METHOD OutputPublish
  VAR_INPUT
    PayloadSize : UDINT;
    PayloadPos : POINTER TO BYTE;  (* be aware, don't use network buffer, IP_CONTROL may change content *)
    TopicSize : UDINT;
    TopicPos : POINTER TO BYTE;  (* be aware, don't use network buffer, IP_CONTROL may change content, must be zero terminated! *)
    MQTT_IN_OUT : POINTER TO MQTT_IN_OUT;
  END_VAR
  VAR
    i : UINT;
    match : TOPIC_MATCH;
    PointerToSplit : POINTER TO SPLIT_TOPIC;
    DataForCallback : CALLBACK_DATA;
  END_VAR
                  //here make everything to give out publish, and test if topic fits to my borders...
CountOutputPublishCalled := CountOutputPublishCalled + 1;
IF MySplitTopic.NewTopic(in:= TopicPos, test := FALSE, SizeOfString:= UDINT_TO_UINT(TopicSize)) = TOPIC_VALID.TOPIC_NOT_VALID THEN
	//topic is not in my borders so throw away data...
	{info 'configure to disconnect?'}
	{ info 'make count var...'}
	CountSplitTopicSizeExceeded := CountSplitTopicSizeExceeded + 1;
	RETURN;
END_IF
//now search the right callback and call it...
PointerToSplit := MySplitTopic.GetSplitTopic();
DataForCallback.Payload := PayloadPos;
DataForCallback.PayloadSize := PayloadSize;
DataForCallback.PayloadString :=PayloadPos;
DataForCallback.TopicOut := TopicPos;
DataForCallback.TopicOutSplit := PointerToSplit;
DataForCallback.PayloadIsString := SubscribeCallbacks[i].ExpectingString;

FOR i := 0 TO CALLBACKS_BUFFER_SIZE - 1 DO
	IF NOT SubscribeCallbacks[i].free THEN
		match := SubscribeCallbacks[i].SplitTopic^.CheckTopicMatchToMe(with:=PointerToSplit);
		IF match = TOPIC_MATCH.TOPIC_MATCHES THEN
			SubscribeCallbacks[i].Callback.PublishRecived(Data:=DataForCallback);
		END_IF
	END_IF
END_FOR


                
END_METHOD

METHOD MergeSplitedPublish
  VAR_INPUT
    MQTT_IN_OUT : POINTER TO MQTT_IN_OUT;
  END_VAR
  VAR
    BytesToMove : UINT;
  END_VAR
                  //move every new data to publish recive buffer untill all data is recived
BytesToMove := TO_UINT(MIN(com.R_BUF.SIZE, SplitPublishLength - SplitPublishBufferSize));
MEM.MemMove(pSource:= ADR(COM.R_BUF.BUFFER), pDestination:= ADR(SplitPublishBuffer[SplitPublishBufferSize]), uiNumberOfBytes:= BytesToMove);
SplitPublishBufferSize := SplitPublishBufferSize + BytesToMove;
IF SplitPublishBufferSize >= SplitPublishLength THEN
	//SplitPublishLock := TRUE;
	PublishSplited := FALSE;
	//ParsePublish will insert string termination if no network buffer
	ParseIncomingPublish(
	MQTT_IN_OUT:= MQTT_IN_OUT, 
	idx:= 0, 
	BufferIn:= SplitPublishBuffer, 
	BufferSize:= SplitPublishBufferSize,
	NetworkBuffer := FALSE);
END_IF
//check if there is more data in buffer --> new packet
IF BytesToMove < COM.R_BUF.SIZE THEN
	//move buffer and set new size...
	MEM.MemMove(pSource:= ADR(COM.R_BUF.BUFFER[BytesToMove]), pDestination:= ADR(COM.R_BUF.BUFFER),
				uiNumberOfBytes:= COM.R_BUF.SIZE - BytesToMove);
	COM.R_BUF.SIZE := COM.R_BUF.SIZE - BytesToMove;
ELSE
	//clear buffer
	COM.R_BUF.SIZE := 0;
	COM.MQTT_RCV_STATE := BYTE#0;//recive zurücksetzten	
END_IF
                
END_METHOD

METHOD Publish : BOOL
  VAR_INPUT
    data : POINTER TO DATA_TO_BROKER;
  END_VAR
  VAR
    i : UINT;
  END_VAR
                  Publish := FALSE;
FOR i := 0 TO MyConstants.QoS_BUFFER_SIZE - 1 DO
	IF OutData[i].step = STEPS_OUT.WAIT_DATA THEN
		OutData[i].InDataFromFb := data;//set Data
		//Pakte id = slot + 1....
		OutData[i].InDataFromFb^.PaketId := i + 1;
		OutgoingPublishOrderIndexCounter := OutgoingPublishOrderIndexCounter + 1;
		OutData[i].PUBLISHOrder :=  OutgoingPublishOrderIndexCounter;
		OutData[i].step := STEPS_OUT.SEND_PUBLSIH;
		CountSendedPublishs := CountSendedPublishs + 1;
		CounterPublishSendForMonitor := CounterPublishSendForMonitor + 1;
		OutData[i].PUBRELRepeatCounter := 0;
		Publish := TRUE;
		EXIT;
	END_IF
END_FOR
                
END_METHOD

METHOD PublishSendDone
  VAR_INPUT
    slot : POINTER TO MQTT_OUT_DATA;
  END_VAR
                  slot^.TimeOutStarted := TRUE;//start Timeout
CASE slot^.InDataFromFb^.MessageQoS OF
	QoS.AtMostOnce:
	//paket gone and bye bye, on QoS 0 
	slot^.InDataFromFb^.SendSucsess := TRUE;
	slot^.step := STEPS_OUT.WAIT_DATA;//can get new data
	QoS.AtLeastOnce:
		slot^.step := STEPS_OUT.WAIT_PUBACK;//wait for ACK
		IF NOT slot^.InDataFromFb^.DUP THEN
			Publishsunacknowledged := Publishsunacknowledged + 1;
		END_IF
	QoS.ExactlyOnce:
		slot^.step := STEPS_OUT.WAIT_PUBREC;//wait for REC
		IF NOT slot^.InDataFromFb^.DUP THEN
			Publishsunacknowledged := Publishsunacknowledged + 1;
		END_IF
END_CASE
                
END_METHOD
END_FUNCTION_BLOCK

FUNCTION_BLOCK HandleSplitTopic
  VAR
    MySplitTopic : SPLIT_TOPIC;
    InitFull : BOOL;
    InitLow : BOOL;
    SplitLength : POINTER TO UINT;  (* this is going to be a pointer to a array of uint to store the string length(and so memmory size) in the string array *)
    TopicsLevel : UINT;
    SplitElementSize : UINT;
    CountSizeExceeded : ULINT;
    TopicsIndexMax : UINT;
    dynMemUsage : POINTER TO UDINT;
  END_VAR

            {info 'TODO test of zeros in strings'}
          

(* use FOR high change OF topic, needs more ram, saves TIME... allocates all memory for the string arrays and strings usefull for often changed topics like recive publish *)
METHOD FullInit : BOOL
  VAR_INPUT
    TopicsLevelInit : UINT;
    SplitElementSizeInit : UINT;
    dynMemUsageInit : POINTER TO UDINT;
  END_VAR
  VAR
    iu : UINT;
  END_VAR
                  dynMemUsage := dynMemUsageInit;
destroy();

InitFull := TRUE;
InitLow := FALSE;

TopicsLevel := TopicsLevelInit;
SplitElementSize := SplitElementSizeInit + 1;//add 1 for trailing 0
IF TopicsLevel > 0 THEN
	TopicsIndexMax := TopicsLevel - 1;
ELSE
	TopicsIndexMax := 0;
END_IF

{warning disable C0033}
//get memory for array of pointer to strings
//MySplitTopic.Topics := SysMem23.SysMemAlloc(dwSize:= TopicsLevel * SIZEOF(MySplitTopic.Topics^));
{info 'semaphore'}
MySplitTopic.Topics := __NEW(POINTER TO STRING, TopicsLevel);
dynMemUsage^ := dynMemUsage^ + TopicsLevel * SIZEOF(MySplitTopic.Topics^);
FOR iu := 0 TO TopicsLevel - 1 DO
	//Get memory for strings
	//MySplitTopic.Topics[iu] := SysMem23.SysMemAlloc(dwSize:= SplitElementSize);	
	{info 'semaphore'}
	MySplitTopic.Topics[iu] := __NEW(BYTE, SplitElementSize);	
	dynMemUsage^ := dynMemUsage^ + SplitElementSize;
END_FOR
{warning restore C0033}

                
END_METHOD

(* use for low change of topic, saves mem, needs time dynamic allocation of memory, usefull for static stopis like compare of subscription topic *)
METHOD LowInit : BOOL
  VAR_INPUT
    TopicsLevelInit : UINT;
    SplitElementSizeInit : UINT;
    dynMemUsageInit : POINTER TO UDINT;
  END_VAR
  VAR
    iu : UINT;
  END_VAR
                  dynMemUsage := dynMemUsageInit;
destroy();
InitFull := FALSE;
InitLow := TRUE;

TopicsLevel := TopicsLevelInit;
SplitElementSize :=SplitElementSizeInit;
IF TopicsLevel > 0 THEN
	TopicsIndexMax := TopicsLevel - 1;
ELSE
	TopicsIndexMax := 0;
END_IF
{warning disable C0033}
//get memory for array of pointer to string 

//MySplitTopic.Topics := SysMem23.SysMemAlloc(dwSize:= TopicsLevel * SIZEOF(MySplitTopic.Topics^));
MySplitTopic.Topics := __NEW(POINTER TO STRING, TopicsLevel);
{info 'semaphore'}
dynMemUsage^ := dynMemUsage^ + TopicsLevel * SIZEOF(MySplitTopic.Topics^);
//get memory for array of length of strings
//SplitLength := SysMem23.SysMemAlloc(dwSize:= TopicsLevel * SIZEOF(SplitLength^));
{info 'semaphore'}
SplitLength := __NEW(POINTER TO STRING, TopicsLevel);
dynMemUsage^ := dynMemUsage^ + TopicsLevel * SIZEOF(SplitLength^);
{warning restore C0033}

                
END_METHOD

METHOD destroy : BOOL
  VAR
    iu : UINT;
  END_VAR
                  GVL_MQTT.ProgNum := PROG_NUM.DESTROY_SPLIT_TOPIC;
IF InitFull THEN
{warning disable C0033}
	FOR iu := 0 TO TopicsLevel - 1 DO
		{info 'semaphore'}
		//SysMem23.SysMemFree(dwAddress:= MySplitTopic.Topics[iu], dwSize:= SplitElementSize);
		__DELETE(MySplitTopic.Topics[iu]);
		dynMemUsage^ := dynMemUsage^ - SplitElementSize;
	END_FOR
	{info 'semaphore'}
	//SysMem23.SysMemFree(dwAddress:= MySplitTopic.Topics, dwSize:= TopicsLevel * SIZEOF(MySplitTopic.Topics^));
	__DELETE(MySplitTopic.Topics);
	dynMemUsage^ := dynMemUsage^ - (TopicsLevel * SIZEOF(MySplitTopic.Topics^));
	InitFull := FALSE;
END_IF

IF InitLow THEN
	DestroyOldSplit();
	{info 'semaphore'}
	//SysMem23.SysMemFree(dwAddress:= MySplitTopic.Topics, dwSize:= TopicsLevel * SIZEOF(MySplitTopic.Topics^));
	__DELETE(MySplitTopic.Topics);
	dynMemUsage^ := dynMemUsage^ - (TopicsLevel * SIZEOF(MySplitTopic.Topics^));
	//SysMem23.SysMemFree(dwAddress:= SplitLength, dwSize:= TopicsLevel * SIZEOF(SplitLength^));
	{info 'semaphore'}
	//SysMem.SysMemFreeData(pMemory:= SplitLength, dwSize:= TopicsLevel * SIZEOF(SplitLength^));
	__DELETE(SplitLength);
	dynMemUsage^ := dynMemUsage^ - (TopicsLevel * SIZEOF(SplitLength^));
	InitLow:= FALSE;
END_IF
{warning restore C0033}
                
END_METHOD

METHOD GetSplitTopic : POINTER TO SPLIT_TOPIC
                  GetSplitTopic := ADR(MySplitTopic);

                
END_METHOD

METHOD FB_Exit : BOOL
  VAR_INPUT
    bInCopyCode : BOOL;  (* TRUE: the exit method is called in order to leave the instance which will be copied afterwards (online change). *)
  END_VAR
                  destroy();

                
END_METHOD

METHOD NewTopic : TOPIC_VALID
  VAR_INPUT
    in : POINTER TO STRING;  (* needs to be 0 terminated! *)
    test : BOOL;  (* check topic, use this for subscriptio, topics from broker should be ok... *)
    SizeOfString : UINT;  (* Size of String, if > 0 then use this size and don't search for 0 *)
  END_VAR
  VAR
    StartSub : DINT;  (* in codesys for mid function first String Position is 1 !!!! devil!!!! don't use anymore, take memmove *)
    i : UINT;
    SplitChar : BYTE;  (* SubCount:UINT; *)
    pt : POINTER TO BYTE;
    UseSize : BOOL;
  END_VAR
                  IF NOT InitFull AND NOT InitLow THEN
	NewTopic := TOPIC_VALID.TOPIC_NOT_VALID;
	RETURN;
END_IF 
DestroyOldSplit();
SplitChar := CommonTypesAndFunctions.GetChar(in:= '/');
GVL_MQTT.ProgNum := PROG_NUM.GetSplitTopic;
IF SizeOfString > 0 THEN
	UseSize := TRUE;
END_IF
pt := in;
WHILE (pt[i] <> 0 AND NOT UseSize) OR (UseSize AND SizeOfString > 0) DO
	SizeOfString := SizeOfString - 1;
	IF pt[i] = SplitChar  THEN
		(*IF ((i - StartSub - 1) > SplitElementSize AND InitFull)THEN
			
		END_IF*)
		IF NOT PushSplitLevel(str:= ADR(in^[StartSub]), len:= i - DINT_TO_UINT(StartSub)) THEN
			CountSizeExceeded := CountSizeExceeded + 1;
			//error pushing split topic
			DestroyOldSplit();
			NewTopic := TOPIC_VALID.TOPIC_NOT_VALID;
			RETURN;
		END_IF
		StartSub := i + 1;//Start Post at next after /
	END_IF
	i := i + 1;
END_WHILE
//get last Topic...
IF NOT (i = StartSub) THEN
	
	PushSplitLevel(str:= ADR(in^[StartSub]), len:= i - DINT_TO_UINT(StartSub));

END_IF
IF pt[i - 1] = SplitChar THEN
	//got one empty level at last
	PushSplitLevel(str:= in, len:= 0);//here str doesnt need to be a valid source
END_IF
IF test THEN
	NewTopic := CheckTopicValid();
	IF NewTopic = TOPIC_VALID.TOPIC_NOT_VALID THEN
		DestroyOldSplit();
	END_IF
ELSE
	NewTopic := TOPIC_VALID.TOPIC_NO_TEST;
END_IF
                
END_METHOD

METHOD PushSplitLevel : BOOL
  VAR_INPUT
    str : POINTER TO STRING;
    len : UINT;
  END_VAR
  VAR
    DynLength : UINT;
  END_VAR
                  //make sure to use no more memmory as allocated
IF (MySplitTopic.ValidFields >=  TopicsIndexMax) OR ((len + 1 > SplitElementSize) AND InitFull) THEN
	PushSplitLevel := FALSE;
	RETURN;
ELSE
	PushSplitLevel := TRUE;
END_IF

IF InitFull THEN
	IF len > 0 THEN
		{'info: TODO: check string length'}
		MEM.MemMove(pSource:= str, pDestination:= MySplitTopic.Topics[MySplitTopic.ValidFields], uiNumberOfBytes:= len);
	END_IF
	MySplitTopic.Topics[MySplitTopic.ValidFields]^[len] := 0;//string limiter
END_IF


IF InitLow THEN
	DynLength := len + 1;
	{warning disable C0033}
	MySplitTopic.Topics[MySplitTopic.ValidFields] := __NEW(BYTE, DynLength);
	//MySplitTopic.Topics[MySplitTopic.ValidFields] := SysMem23.SysMemAlloc(dwSize:= DynLength);
	dynMemUsage^ := dynMemUsage^ + DynLength;
	{warning restore C0033}
	IF len > 0 THEN
		MEM.MemMove(pSource:= str, pDestination:= MySplitTopic.Topics[MySplitTopic.ValidFields], uiNumberOfBytes:= len);
	END_IF
	SplitLength[MySplitTopic.ValidFields] := DynLength;
	MySplitTopic.Topics[MySplitTopic.ValidFields]^[DynLength - 1] := 0;//string limiter
END_IF

MySplitTopic.ValidFields := MySplitTopic.ValidFields + 1;
                
END_METHOD

METHOD DestroyOldSplit
  VAR
    di : DINT;
  END_VAR
                  IF InitLow THEN
	FOR di := 0 TO MySplitTopic.ValidFields - 1 DO
{warning disable C0033}
{info 'semaphore'}
		//SysMem23.SysMemFree(dwAddress:= MySplitTopic.Topics[di], dwSize:= SplitLength[di]);
		__DELETE(MySplitTopic.Topics[di]);
		
		dynMemUsage^ := dynMemUsage^ - SplitLength[di];
{warning restore C0033}		
	END_FOR
END_IF

MySplitTopic.ValidFields := 0;
                
END_METHOD

(* Instance needs to be subscription topic *)
METHOD CheckTopicMatchToMe : TOPIC_MATCH
  VAR_INPUT
    with : POINTER TO SPLIT_TOPIC;  (* topic to compare with, here the topic from broker *)
  END_VAR
  VAR
    i : UINT;
    pt : POINTER TO BYTE;
    wildcard : BYTE;
  END_VAR
                  wildcard := CommonTypesAndFunctions.GetChar(in:= '#');
FOR i := 0 TO MIN(MySplitTopic.ValidFields - 1, with^.ValidFields - 1) DO
	pt := MySplitTopic.Topics[i]; 
	IF pt^ = wildcard THEN
		//from here its mine
		CheckTopicMatchToMe := TOPIC_MATCH.TOPIC_MATCHES;
		RETURN;
	END_IF
	IF NOT CheckTopicLevel(s1:= with^.Topics[i] , s2:= MySplitTopic.Topics[i]) THEN
		CheckTopicMatchToMe := TOPIC_MATCH.TOPIC_DONT_MATCHES;
		RETURN;
	END_IF  
END_FOR
//if here and there are further topics then its note mine
IF MySplitTopic.ValidFields = with^.ValidFields THEN
	CheckTopicMatchToMe := TOPIC_MATCH.TOPIC_MATCHES;
	RETURN;
END_IF
pt := ADR(MySplitTopic.Topics[i]);
IF MySplitTopic.ValidFields > with^.ValidFields AND 
	pt^ = wildcard THEN
	//check last Subscription topic if '#'
	CheckTopicMatchToMe := TOPIC_MATCH.TOPIC_MATCHES;
ELSE
	CheckTopicMatchToMe := TOPIC_MATCH.TOPIC_DONT_MATCHES;
END_IF
                
END_METHOD

METHOD CheckTopicValid : TOPIC_VALID
  VAR
    i : UINT;
  END_VAR
                  FOR i := 0 TO MySplitTopic.ValidFields - 1 DO
	IF (CommonTypesAndFunctions.find(STR1:= MySplitTopic.Topics[i], STR2:= ADR('#')) >= 0) AND (CommonTypesAndFunctions.len(STR:= MySplitTopic.Topics[i]) > 1) THEN
		//error # within topic
		CheckTopicValid := TOPIC_VALID.TOPIC_NOT_VALID;
		RETURN;
		
	END_IF
	IF (CommonTypesAndFunctions.find(STR1:= MySplitTopic.Topics[i], STR2:= ADR('+')) >= 0) AND (CommonTypesAndFunctions.len(STR:= MySplitTopic.Topics[i]) > 1) THEN
		//error + within topic
		CheckTopicValid := TOPIC_VALID.TOPIC_NOT_VALID;
		RETURN;
	END_IF
		IF (CommonTypesAndFunctions.find(STR1:= MySplitTopic.Topics[i], STR2:= ADR('#')) >= 0) AND (i <> MySplitTopic.ValidFields - 1) THEN
		//error # not at lowest topic
		CheckTopicValid := TOPIC_VALID.TOPIC_NOT_VALID;
		RETURN;
	END_IF
END_FOR
CheckTopicValid := TOPIC_VALID.TOPIC_VALID;

                
END_METHOD
END_FUNCTION_BLOCK

FUNCTION_BLOCK InsertSplitPayload
  VAR_INPUT
    payload : POINTER TO BYTE;  (* payload to insert.... *)
    len : UDINT;  (* length of payload *)
    buff : POINTER TO BYTE;  (* address to buffer *)
    pos : UINT;  (* Start to insert *)
    size : UINT;  (* size of buffer *)
  END_VAR
  VAR_OUTPUT
    state : INSERT_SPLIT_RETURN;
    new_pos : UINT;
  END_VAR
  VAR
    step : INT;
    akt_pos : UDINT;
  END_VAR
  VAR_TEMP
    bytes_to_send : UINT;
  END_VAR

            //always make my output valid
new_pos := pos;

IF step = 0 THEN
	step := 10;//start insert...
END_IF

//don't use case, so save a cyle...
IF step = 10 THEN
	//evaluate if we have to split payload....
	IF size - pos < len THEN
		step := 20;
		akt_pos := 0;
	ELSE
		//here no split needed
		MEM.MemMove(pSource:= payload, pDestination:= ADR(buff[new_pos]), uiNumberOfBytes:= UDINT_TO_UINT(len));
		new_pos := UDINT_TO_UINT(new_pos + len);//new pos for output
		state := INSERT_SPLIT_RETURN.INSERT_DONE;
		step := 0;
	END_IF
END_IF

IF step = 20 THEN
	//now do split payload...
	bytes_to_send := UDINT_TO_UINT(MIN(size - new_pos, len - akt_pos));
	MEM.MemMove(pSource:= ADR(payload[akt_pos]), pDestination:= ADR(buff[new_pos]), uiNumberOfBytes:= bytes_to_send);
	akt_pos := akt_pos + bytes_to_send;
	new_pos := new_pos +  bytes_to_send;
	IF akt_pos + 1 >= len THEN
		//send done
		state := INSERT_SPLIT_RETURN.INSERT_DONE;
		step := 0;
	ELSE
		state := INSERT_SPLIT_RETURN.INSERT_PENDING;
	END_IF
END_IF

          

METHOD reset
                  step := 0;
                
END_METHOD
END_FUNCTION_BLOCK

FUNCTION_BLOCK InsertSplitTopic
  VAR_INPUT
    topic : POINTER TO STRING;  (* topic to insert.... *)
    len : UINT;  (* length of topic *)
    buff : POINTER TO BYTE;  (* address to buffer *)
    pos : UINT;  (* Start to insert *)
    size : UINT;  (* size of buffer *)
  END_VAR
  VAR_OUTPUT
    state : INSERT_SPLIT_RETURN;
    new_pos : UINT;
  END_VAR
  VAR
    step : INT;
    akt_pos : UINT;
  END_VAR
  VAR_TEMP
    bytes_to_send : UINT;
  END_VAR

            //always make my output valid
new_pos := pos;

IF step = 0 THEN
	step := 10;//start insert...
END_IF

//don't use case, so save a cyle...
IF step = 10 THEN
	//check if buffer size is enogh for header
	IF size - new_pos < 2 THEN
		state := INSERT_SPLIT_RETURN.INSERT_ERROR;
		RETURN;
	END_IF
	buff[new_pos]:= OSCAT_BASIC.BYTE_OF_DWORD(in:= len, N:= 1);
	buff[new_pos+1]:= OSCAT_BASIC.BYTE_OF_DWORD(in:= len, N:= 0);
	new_pos := new_pos + 2;
	step := 20;
END_IF

IF step = 20 THEN
	//evaluate if we have to split topic....
	IF size - pos < len THEN
		step := 30;
		akt_pos := 0;
	ELSE
		//here no split needed
		MEM.MemMove(pSource:= topic, pDestination:= ADR(buff[new_pos]), uiNumberOfBytes:= len);
		new_pos := new_pos + len;//new pos for output
		state := INSERT_SPLIT_RETURN.INSERT_DONE;
		step := 0;
	END_IF
END_IF

IF step = 30 THEN
	//now do split topic...
	bytes_to_send := MIN(size - new_pos, len - akt_pos);
	MEM.MemMove(pSource:= ADR(topic^[akt_pos]), pDestination:= ADR(buff[new_pos]), uiNumberOfBytes:= bytes_to_send);
	akt_pos := akt_pos + bytes_to_send;
	new_pos := new_pos +  bytes_to_send;
	IF akt_pos + 1 >= len THEN
		//send done
		state := INSERT_SPLIT_RETURN.INSERT_DONE;
		step := 0;
	ELSE
		state := INSERT_SPLIT_RETURN.INSERT_PENDING;
	END_IF
END_IF

          

METHOD reset
                  step := 0;
                
END_METHOD
END_FUNCTION_BLOCK

FUNCTION_BLOCK MQTT_CONTROL
  VAR_IN_OUT
    COM : MQTT_COM;
    INFO : MQTT_INFO;
  END_VAR
  VAR
    IP_C : IP_C;
    URL_DATA : url;
    IPC : CommonTypesAndFunctions.IP_CONTROL_TLS;  (* DNS_CLIENT : DNS_CLIENT; *)
    sResultIP : STRING;  (* IP-Address behind hostname *)
    rtsResult : RTS_IEC_RESULT;
    step : INT;
    snd_step : INT;
    TON_WAIT : OSCAT_BASIC.TON;
    last_step : INT;
    idx1 : UINT;
    connectToLocalhost : BOOL;
    staticIP : BOOL;
    timeout1 : TIME;  (* idx2 : INT; idx3 : INT; dw_tmp : DWORD; *)
    timeout2 : TIME;
    ip_c_red_disable : BOOL;
    remaining_length : UINT;
    domainLowercase : STRING(255);
    nop : INT;  (* LOG_MSG : LOG_MSG; _debug_enable : BOOL := TRUE; *)
    S_BUF : NETWORK_BUFFER;  (* ****************************************************************************** here all TLS Stuff *)
    R_BUF : NETWORK_BUFFER;
    TLSConnection : RTS_IEC_HANDLE;  (* ****************************************************************************** RTSResult: RTS_IEC_RESULT; *)
  END_VAR
  VAR_TEMP
    WillTopic : STRING(255);
  END_VAR

            IF com.ERROR_C <> 0 THEN
 step := step;
END_IF 
//init Pointers


CASE step OF

00:	IF COM.MQTT_CON THEN

		timeout1 := MAX(T#10S,COM.TIMEOUT);
		timeout2 := timeout1 + T#1s;
		INFO.MQTT_ERROR := '';
		COM.ERROR_C := DWORD#0;
		COM.ERROR_T := BYTE#0;
		URL_DATA := STRING_TO_URL(STR:=COM.MQTT_URL,DEFAULT_PROTOCOL:='',DEFAULT_PATH:='/');
		domainLowercase := OSCAT_BASIC.LOWERCASE(str:=URL_DATA.DOMAIN );
		IF  CommonTypesAndFunctions.StrEqualsAtStart(str1:= ADR(domainLowercase), str2:= ADR('localhost')) THEN
			connectToLocalhost := TRUE;
		ELSE
			connectToLocalhost := FALSE;
		END_IF
		IF OSCAT_NETWORK.IP4_DECODE(str:= URL_DATA.DOMAIN) > 0 THEN
			sResultIP := URL_DATA.DOMAIN;
			staticIP := TRUE;
		ELSE
			staticIP := FALSE;
		END_IF
		IF connectToLocalhost OR staticIP THEN
			//jump to connect
			step := 20;
		ELSE
			//get ip by dns
			step := 10;
		END_IF
	END_IF;

10:
	IF CommonTypesAndFunctions.ResolveIPAddr(sHost:= URL_DATA.DOMAIN, sIPResult:= ADR(sResultIP)) = CmpErrors.Errors.ERR_OK THEN
		step := 20;
	ELSE
		step := 980;
	END_IF

20:	(* MQTT Steuerkanal einrichten *)
	IF URL_DATA.PORT = WORD#0 THEN
		URL_DATA.PORT := WORD#1883; (* Standard Port *)
	END_IF;
	IP_C.C_PORT := URL_DATA.PORT; (* Portnummer eintragen *)
	IF connectToLocalhost THEN
		IP_C.C_IP := IP4_DECODE('127.0.0.1'); (* IP eintragen, localhost *)
	ELSE
		IP_C.C_IP := IP4_DECODE(sResultIP); (* IP eintragen *)
	END_IF
  	
	IP_C.C_MODE := BYTE#0; (* Mode: TCP+ACTIV+PORT *)
  	IP_C.TIME_RESET := TRUE; (* Zeitueberwachung rücksetzen *)
  	IP_C.C_ENABLE := TRUE; (* Verbindungsaufbau freigeben *)
  	IP_C.R_OBSERVE := FALSE; (* Empfangsueberwachung *)
	COM.R_BUF.SIZE := UINT#0;
	COM.MQTT_RCV_STATE := BYTE#0;
	step := 30;
	

30:	 IF IP_C.C_STATE = BYTE#255 THEN
		COM.S_BUF.BUFFER[0] := MESSAGETYPE.CONNECT;
		COM.S_BUF.BUFFER[1] := 0;//Header length, cal at least
		COM.S_BUF.BUFFER[2] := 0;//Variable Header length
		COM.S_BUF.BUFFER[3] := 4;//Variable Header length
		COM.S_BUF.BUFFER[4] := OSCAT_BASIC.CODE(STR:= 'M', POS:= 1);//Protokoll name
		COM.S_BUF.BUFFER[5] := OSCAT_BASIC.CODE(STR:= 'Q', POS:= 1);//Protokoll name
		COM.S_BUF.BUFFER[6] := OSCAT_BASIC.CODE(STR:= 'T', POS:= 1);//Protokoll name
		COM.S_BUF.BUFFER[7] := OSCAT_BASIC.CODE(STR:= 'T', POS:= 1);//Protokoll name
		COM.S_BUF.BUFFER[8] := 4; //Protokoll Level
		COM.S_BUF.BUFFER[9] := 2#00110110;//Connect flags
							   //|||||||+-Reserved
							   //||||||+--Clean Session
							   //|||||+---Will Flag
							   //|||++----Will QoS
							   //||+------Will Retain
							   //|+-------Password Flag
							   //+--------UserNameFlag
		COM.S_BUF.BUFFER[10] := OSCAT_BASIC.BYTE_OF_DWORD(in:= MyConstants.KEEP_ALIVE_TIME, N:= 1);//keep alive MSB
		COM.S_BUF.BUFFER[11] := OSCAT_BASIC.BYTE_OF_DWORD(in:= MyConstants.KEEP_ALIVE_TIME, N:= 0);//keep alive LSB
		//idx1 points to next free byte
		//now put in client id 
		idx1 := InsertStringToBufferAndLength(Str:= ADR(COM.CLIENT_ID), buff:= ADR(COM.S_BUF.BUFFER), pos:= 12(*, size:= OSCAT_NETWORK.Constants.NETWORK_BUFFER_LONG_SIZE*));
		//now put in will topic
		WillTopic := Standard.CONCAT(STR1:= COM.CLIENT_ID, STR2:= Standard.CONCAT(STR1:= '/', STR2:= COM.CLIENT_WILL_TOPIC));
		idx1 := InsertStringToBufferAndLength(Str:= ADR(WillTopic), buff:= ADR(COM.S_BUF.BUFFER), pos:= idx1(*, size:= OSCAT_NETWORK.Constants.NETWORK_BUFFER_LONG_SIZE*));
		//now put in will message
		//IF Standard.LEN(STR:= COM.CLIENT_WILL_MESSAGE_DEAD) > 0 THEN
		idx1 := InsertStringToBufferAndLength(Str:= ADR(COM.CLIENT_WILL_MESSAGE_DEAD), buff:= ADR(COM.S_BUF.BUFFER), pos:= idx1(*, size:= OSCAT_NETWORK.Constants.NETWORK_BUFFER_LONG_SIZE*));
		//END_IF
		//if user is given, set user bit an insert username
		IF Standard.LEN(STR:= COM.BROKER_USER) > 0 THEN
			COM.S_BUF.BUFFER[8] := COM.S_BUF.BUFFER[8] OR 2#10000000;
			//now put in user name
			idx1 := InsertStringToBufferAndLength(Str:= ADR(COM.BROKER_USER), buff:= ADR(COM.S_BUF.BUFFER), pos:= idx1(*, size:= OSCAT_NETWORK.Constants.NETWORK_BUFFER_LONG_SIZE*));
		END_IF
		//if password is given, set password bit an insert username
		IF Standard.LEN(STR:= COM.BROKER_PASSWORD) > 0 THEN
			COM.S_BUF.BUFFER[8] := COM.S_BUF.BUFFER[8] OR 2#1000000;
			//now put in user name
			idx1 := InsertStringToBufferAndLength(Str:= ADR(COM.BROKER_PASSWORD), buff:= ADR(COM.S_BUF.BUFFER), pos:= idx1(*, size:= OSCAT_NETWORK.Constants.NETWORK_BUFFER_LONG_SIZE*));
		END_IF
		//now cal packet lengt and insert remaining legth
		remaining_length := idx1 - 2;
		DoRemainingLength(buffer:= ADR(com.S_BUF.BUFFER), RemainingLength:= remaining_length);
		//now send data
		COM.S_BUF.SIZE := idx1;
		step := 40;//wait for CONNACK
	END_IF
	
		
40:	//IF COM.MQTT_RCV_STATE = BYTE#1 THEN//recived packet
	IF COM.R_BUF.SIZE > 0 THEN//recived packet
		IF COM.R_BUF.BUFFER[0] <> MESSAGETYPE.CONNACK THEN
			step := 700;//close connection
		ELSE//get connack packet
			IF COM.R_BUF.BUFFER[3] = 0 THEN
				//connection accepted
				INFO.MQTT_CONNECTED := TRUE;
				COM.R_BUF.SIZE := 0;
				COM.MQTT_RCV_STATE := BYTE#0;
				step := 300;
			ELSE
				step := 700;//close connection
			END_IF
		END_IF
		
	END_IF


(* ================================================== *)

300:	step := UINT_TO_INT(SEL(COM.MQTT_CON,700,310)); (* Schritt-Selektion *)

310:	step := 300; (* dummy step *)

(* ================================================== *)

700: (* COM_QUIT *)
	//INFO.MQTT_CONNECTED := FALSE;
	IF COM.MQTT_ABORT THEN
		step := 980;//close without disconnect packet
		COM.MQTT_ABORT := FALSE;
	ELSE
		COM.S_BUF.BUFFER[0] := MESSAGETYPE.DISCONNECT; (* 0x01 COM_QUIT mqtt_close *)
		COM.S_BUF.BUFFER[1] := 0;
		COM.S_BUF.SIZE := UINT#2; (* Sendelänge eintragen *)
		
		ip_c_red_disable := TRUE;
		step := 710;
	END_IF
710:	IF COM.S_BUF.SIZE = BYTE#0 THEN (* letztes Paket gesendet?*)
		step := 980;
	END_IF;

(* ================================================== *)

980:IP_C.C_ENABLE := FALSE; (* MQTT Steuerkanal schliessen *)
	ip_c_red_disable := FALSE;
	INFO.MQTT_CONNECTED := FALSE;
	COM.MQTT_CON := FALSE;
	COM.S_BUF.SIZE := UINT#0;
	COM.R_BUF.SIZE := UINT#0;
	snd_step := 0;
	step := 990;
	(*####################  DEBUG-MESSAGE  ###################################*)
	(*IF _debug_enable THEN
		LOG_CL.NEW_MSG := 'QUIT: ERROR CODE >~1< TYPE >~2<';
		LOG_CL.PRINTF[1] := DWORD_TO_STRH(COM.ERROR_C);
		LOG_CL.PRINTF[2] := BYTE_TO_STRING(COM.ERROR_T);
		LOG_MSG();
	END_IF;*)
	(*########################################################################*)

990:IF IP_C.C_STATE = BYTE#0 THEN
		step := 0;
	END_IF;

END_CASE;

(* ++++++++++++++++++++++++++++++++++++++++++++++++++++++++++ *)
IF step > 40 THEN
	IF COM.R_BUF.SIZE >= UINT#1 THEN (* Daten wurden empfangen ? neue kommunikation*)
		
		COM.MQTT_RCV_STATE := BYTE#1;
		
	END_IF;
END_IF;
(* automatisches Datensenden *)

CASE snd_step OF

00:	IF step > 40 THEN
	
		IF COM.S_BUF.SIZE > UINT#0 THEN
	
		    (*####################  DEBUG-MESSAGE  ###################################*)
	        (*IF _debug_enable THEN
	          LOG_CL.NEW_MSG := 'SND: size >~1<';
	          LOG_CL.PRINTF[1] := UINT_TO_STRING(COM.S_BUF.SIZE);
	          LOG_MSG();
	        END_IF;*)
	        (*########################################################################*)

			snd_step := 10;
		END_IF;		
	END_IF;

10:	IF COM.S_BUF.SIZE = UINT#0 THEN (* warten bis alle daten gesendet sind *)
		snd_step := 0;
	END_IF;

END_CASE;

(* Globale Fehlerbehandlung für Haupt-Routine *)
IF COM.ERROR_T = BYTE#0 AND step > 20 THEN (* noch kein Fehler gespeichert und Hauptroutine aktiv *)
	IF IP_C.ERROR > DWORD#0 AND IP_C.C_ENABLE AND NOT IP_C.TIME_RESET THEN  (* IP Control *)
		IF ip_c_red_disable = FALSE OR IP_C.ERROR <> DWORD#16#FD000000 THEN
			COM.ERROR_C := IP_C.ERROR;
			COM.ERROR_T := BYTE#2;
			step := 980;
		END_IF;
	END_IF;
END_IF;

IF TON_WAIT.Q THEN (* Ablaufstörung - Schrittkette *)
	COM.ERROR_C := INT_TO_DWORD(step); (* aktuellen Schritt eintragen *)
	COM.ERROR_T := BYTE#5;
	step := 980;
END_IF;

(* ######################################################## *)

//DNS_CLIENT(IP_C:=IP_C, S_BUF:=COM.S_BUF, R_BUF:=COM.R_BUF, DOMAIN:=URL_DATA.DOMAIN, IP4_DNS:= COM.DNS_IP4, ACTIVATE:=step=10); (* DNS-Client *)
IPC(IP:= DWORD#0, PORT:= WORD#0 , TIME_OUT:= timeout1, IP_C:= IP_C, S_BUF:= COM.S_BUF, R_BUF:= COM.R_BUF, TLS_CONFIG_IN := COM.TLS_CONFIG, useTls:= COM.TLS); (* MQTT Steuerkanal *)

TON_WAIT(IN:=step = last_step AND step > 0,PT:=timeout2);
last_step := step;


(* revision history


*)
          
END_FUNCTION_BLOCK

FUNCTION_BLOCK MQTTBase
  VAR
    MQTT_IN_OUT : POINTER TO MQTT_IN_OUT;
    DbPointerIo : BOOL;  (* Set to true if get DB Pointer *)
    TokenRequested : BOOL;
    RTrig : r_trig;
    COM_CONFIG : COM_CONFIG;  (* config for boot up *)
  END_VAR

            IF not DbPointerIo THEN RETURN; END_IF
MQTT_IN_OUT^.FB_NO_AUTO := MQTT_IN_OUT^.FB_NO_AUTO + 1;
          

METHOD SetMqttInOut : INT
  VAR_INPUT
    MQTT_IN_OUT : POINTER TO MQTT_IN_OUT;
  END_VAR
                  THIS^.MQTT_IN_OUT := MQTT_IN_OUT;
DbPointerIo := TRUE;
                
END_METHOD

METHOD RequestToken
  VAR_INPUT
    request : BOOL;
  END_VAR
                  RTrig(CLK:= request);
//IF RTrig.Q THEN
IF request THEN
	TokenRequested := TRUE;
END_IF
                
END_METHOD

METHOD ReleaseToken
                  IF MQTT_IN_OUT^.FB_NO_AUTO =  MQTT_IN_OUT^.FB_NO_AUTO_TOKEN THEN
	MQTT_IN_OUT^.FB_NO_AUTO_TOKEN := MQTT_IN_OUT^.FB_NO_AUTO_TOKEN + 1;
END_IF
TokenRequested := FALSE;
                
END_METHOD
END_FUNCTION_BLOCK

(* be aware, don't change payload an topic until send is done!!! *)
FUNCTION_BLOCK MQTTPublish EXTENDS MQTTBase
  VAR_INPUT
    Topic : POINTER TO STRING;  (* here your topic *)
    PayloadString : POINTER TO STRING;  (* here the payload String *)
    PublishAsString : BOOL;  (* set this to true to publish a string, else the data is expected on Payload *)
    Payload : POINTER TO BYTE;  (* binary payload *)
    PayloadLength : UDINT;  (* length of binary payload *)
    QoSIn : QoS;  (* QoS Level *)
    MRetain : BOOL;  (* Message is retain? *)
    send : BOOL;  (* send on positiv edge, be aware, don't change payload an topic until send is done!!! *)
  END_VAR
  VAR_OUTPUT
    done : BOOL;  (* sucsessfull transmittet *)
    sendActive : BOOL;  (* trying to send *)
    SendTimeout : BOOL;  (* Timout of sending while connection io --> to much load *)
    CountSend : ULINT;  (* count of publish send sucsessfull *)
  END_VAR
  VAR
    requestToSend : BOOL;
    TriggerEdge : Standard.R_TRIG;
    WasSendet : BOOL;  (* paket gone out *)
    TimeToResponse : CAA.TICK;
    LastSend : CAA.TICK;
    MyOutData : DATA_TO_BROKER;
    DUP : BOOL;  (* retry bit *)
    SendTimeOutTime : ton;  (* timeout timer *)
  END_VAR

            SUPER^();
//if not config, then leave, do this after super so we calc correct FB numbers
IF NOT DbPointerIo THEN RETURN; END_IF;
GVL_MQTT.ProgNum := PROG_NUM.Publish;
TriggerEdge(CLK:= send AND NOT requestToSend AND MQTT_IN_OUT^.BROKER_CONNECTED);

IF NOT MQTT_IN_OUT^.BROKER_CONNECTED THEN
	//no connection, reset
	WasSendet := FALSE;
	IF requestToSend THEN
		DUP := TRUE;
	END_IF
	
END_IF

done := FALSE;

IF TriggerEdge.Q THEN
	requestToSend := TRUE;
END_IF

IF requestToSend AND NOT WasSendet THEN
	//try to publish
	MyOutData.PaketData.MqttTopicLength := CommonTypesAndFunctions.LEN(Topic);
	//don't sent zero lengt topics...
	IF  MyOutData.PaketData.MqttTopicLength > 0 THEN
		MyOutData.PaketData.FbId := MQTT_IN_OUT^.FB_NO_AUTO;
		MyOutData.PaketData.MessageType := MESSAGETYPE.PUBLISH;
		MyOutData.PaketData.MessageRetain := MRetain;
		MyOutData.PaketData.MessageQoS := QoSIn;
		IF PublishAsString THEN
			MyOutData.PaketData.MqttPayloadLength := CommonTypesAndFunctions.LEN(PayloadString);
			MyOutData.PaketData.MqttPayload := PayloadString;
		ELSE
			MyOutData.PaketData.MqttPayloadLength := PayloadLength;
			MyOutData.PaketData.MqttPayload := Payload;
		END_IF
		MyOutData.PaketData.MqttTopic := Topic;
		MyOutData.PaketData.DUP := DUP;
		//WasSendet := TRUE;
		LastSend := TICKS.GetTick(xDummy:= TRUE);
	ELSE
		{info 'check if we want to diplay topic error'}
		;
	END_IF
	IF MQTT_IN_OUT^.handleFB^.Publish(data:=ADR(MyOutData)) THEN
		WasSendet := TRUE;
	ELSE
		WasSendet := FALSE;
	END_IF
END_IF


IF MyOutData.PaketData.SendSucsess THEN //sucsses set by HANDLE_MQTT
	MyOutData.PaketData.SendSucsess := FALSE;
	//paket away...
	WasSendet := FALSE;
	requestToSend := FALSE; 
	done := TRUE;
	DUP := FALSE;
	MyOutData.PaketData.DUP := FALSE;
	TimeToResponse := TICKS.GetTick(xDummy:= TRUE) - LastSend;
	CountSend := CountSend + 1;
END_IF

SendTimeOutTime(IN:= requestToSend, PT:= MyConstants.SENDING_TIMEOUT);
SendTimeout := SendTimeOutTime.Q;

sendActive := requestToSend;
          
END_FUNCTION_BLOCK

FUNCTION_BLOCK MQTTPushover
  VAR_INPUT
    Data : POINTER TO PUSHOVER_DATA;
    MQTT_IN_OUT : POINTER TO MQTT_IN_OUT;
    CountData : UINT;
    MQTTTopic : POINTER TO STRING;
  END_VAR
  VAR
    i : UINT;
    HaveToPush : BOOL;
    Publish : MQTTPublish;
    init : BOOL;
    PushedElement : UINT;
    SendFree : BOOL;
    hit : BOOL;  (* at least one message to push *)
    hitIndex : UINT;
    SendString : STRING(500);  (* build like 'Topic(n(x)):x, Payload(n(x):x, Prio:x, Sound:x' *)
    tmpString : STRING;
  END_VAR

            IF NOT init THEN
	
	init := TRUE;
	Publish.SetMqttInOut(MQTT_IN_OUT:= MQTT_IN_OUT);
END_IF
hit := FALSE;
HaveToPush := FALSE;
FOR i := 0 TO CountData - 1 DO
	IF Data[i].IsConfig THEN
		Data[i].R_T(CLK:=Data[i].Trigger^ XOR Data[i].Negate);
		IF Data[i].R_T.Q THEN
			Data[i].NeedToPush := TRUE;
		END_IF
		IF Data[i].NeedToPush THEN
			HaveToPush := TRUE;
		END_IF
		IF HaveToPush and NOT hit THEN
			hit := TRUE;
			hitIndex := i;
		END_IF
	END_IF
END_FOR

IF Publish.done THEN
	SendFree := TRUE;
END_IF


IF HaveToPush AND SendFree THEN
	SendFree := FALSE;
	//now build message
	SendString := 'Topic(';
	//add topic length
	tmpString := TO_STRING(len(Data[hitIndex].Topic^));
 	CommonTypesAndFunctions.concat(s1:= ADR(SendString), S2:=ADR(tmpString));
	//add '):'
	CommonTypesAndFunctions.concat(s1:= ADR(SendString), S2:=ADR('):'));
	//add topic
	CommonTypesAndFunctions.concat(s1:= ADR(SendString), S2:=Data[hitIndex].Topic);
	//add fixtext
	CommonTypesAndFunctions.concat(s1:= ADR(SendString), S2:=ADR(', Payload('));
	//add payload length
	tmpString := TO_STRING(len(Data[hitIndex].Payload^));
 	CommonTypesAndFunctions.concat(s1:= ADR(SendString), S2:=ADR(tmpString));
	//add '):'
	CommonTypesAndFunctions.concat(s1:= ADR(SendString), S2:=ADR('):'));
	//add topic
	CommonTypesAndFunctions.concat(s1:= ADR(SendString), S2:=Data[hitIndex].Payload);
	//add fixtext
	CommonTypesAndFunctions.concat(s1:= ADR(SendString), S2:=ADR(', Prio:'));
	//add prio
	tmpString := TO_STRING(Data[hitIndex].Prio);
 	CommonTypesAndFunctions.concat(s1:= ADR(SendString), S2:=ADR(tmpString));
	//add fixtext
	CommonTypesAndFunctions.concat(s1:= ADR(SendString), S2:=ADR(', Sound:'));
	//add prio
	tmpString := TO_STRING(Data[hitIndex].Sound);
 	CommonTypesAndFunctions.concat(s1:= ADR(SendString), S2:=ADR(tmpString));
	//done
	Data[hitIndex].NeedToPush := FALSE;
	//now send
	
END_IF

Publish(
	Topic:= MQTTTopic, 
	PayloadString:= adr(SendString), 
	PublishAsString:= TRUE, 
	QoSIn:= QoS.ExactlyOnce, 
	MRetain:= true, 
	send:= NOT SendFree);
          
END_FUNCTION_BLOCK

FUNCTION_BLOCK MQTTState
  VAR
    State : POINTER TO BOOL;
    Topic : POINTER TO STRING;
    StateName : POINTER TO STRING;
    StateValueOn : POINTER TO STRING;
    StateValueOff : POINTER TO STRING;
    InitDone : BOOL;
    Send : BOOL;
    SendDone : BOOL;
    RequestToSendOn : BOOL;
    RequestToSendOff : BOOL;
    publish : MQTTPublish;
    PayloadTemplate : STRING(255);
    Payload : STRING(255);
    QoS : QoS;
    RetainMqtt : BOOL;
    RT : R_TRIG;  (* SendBlock: BOOL; *)
    FT : F_TRIG;
  END_VAR

            //need to call publish here because of FB nums
publish(
	Topic:= Topic, 
	PayloadString:= ADR(Payload), 
	PublishAsString:= TRUE, 
	QoSIn:= QoS, 
	MRetain:= RetainMqtt, 
	send:= Send, 
	done=> SendDone);

IF NOT InitDone THEN RETURN; END_IF
RT(CLK:= State^);
FT(CLK:= State^);

IF RT.Q THEN
	RequestToSendOn := TRUE;
END_IF

IF FT.Q THEN
	RequestToSendOff := TRUE;
END_IF

IF RequestToSendOn AND NOT send THEN
	//send on
	send:= TRUE;
	Payload := PayloadTemplate;
	CommonTypesAndFunctions.concat(s1:= ADR(Payload), s2:= StateValueOn);
	RequestToSendOn := FALSE;
END_IF

IF RequestToSendOff AND NOT send THEN
	//send on
	send:= TRUE;
	Payload := PayloadTemplate;
	CommonTypesAndFunctions.concat(s1:= ADR(Payload), s2:= StateValueOff);
	RequestToSendOff := FALSE;
END_IF

IF SendDone THEN
	Send := FALSE;
END_IF
          

METHOD Init
  VAR_INPUT
    State : POINTER TO BOOL;  (* pointer to state *)
    Topic : POINTER TO STRING;  (* topic name *)
    StateName : POINTER TO STRING;  (* valuve name, placed with ':' bevor value *)
    StateValueOn : POINTER TO STRING;
    StateValueOff : POINTER TO STRING;
    MQTT_IN_OUT : POINTER TO MQTT_IN_OUT;  (* Pointer MQTTT exchange strucure *)
    QoS : QoS;  (* QoS lewvel of publish *)
    RetainMqtt : BOOL;  (* message should be ratained? *)
  END_VAR
                  publish.SetMqttInOut(MQTT_IN_OUT := MQTT_IN_OUT);
THIS^.State := State;
THIS^.Topic := Topic;
THIS^.StateName := StateName;
THIS^.StateValueOff := StateValueOff;
THIS^.StateValueOn := StateValueOn;
THIS^.PayloadTemplate := StateName^;
//don't ad ':' if no name is given
IF NOT THIS^.PayloadTemplate[0] = 0 THEN
	CommonTypesAndFunctions.concat(s1:= ADR(THIS^.PayloadTemplate), s2:= ADR(':'));
ELSE
	PayloadTemplate[0] := 0;
END_IF

InitDone := TRUE;
THIS^.RetainMqtt := RetainMqtt;
THIS^.QoS := QoS;

                
END_METHOD
END_FUNCTION_BLOCK

(* use this to subscribe to a topic, if the topic you want to subscribe isn't valid you get an error on output SubscribeFail, subscribing now uses callbacks for recived publsih packets. you have to pass a FB instance which implements the "MQTT_SUBSCRIBE_CALLBACK" interface. after reciving a matching topic to the subscription topic, the method PublisRecived() of the FB is called. The call passes all needed information to the callback. in the called method you can differ the topic or payload more finer if needed. See the ListAllValueCallback() and ListStringCallback for example. they using a list to the exact topic. So you can subscribe to a topic with wildcard or fix topic with coded payload, and the list FBs doing the fine stuff. *)
FUNCTION_BLOCK MQTTSubscribe EXTENDS MQTTBase
  VAR_INPUT
    Subscribe : BOOL;  (* set to true to subscribe, set to false to unsubscribe *)
    Topic : POINTER TO STRING;  (* your topic string *)
    QoSSubscribe : QoS;  (* QoS level *)
    ExpectingString : BOOL;  (* set to true is you want an string as output, if so you get the String on PayloadString, else you get binary data on payload *)
    Callback : MQTT_SUBSCRIBE_CALLBACK;  (* callback FB *)
  END_VAR
  VAR_OUTPUT
    SubscribeDone : BOOL;
    SendTimeout : BOOL;  (* Timout of sending(subscribe paket) while connection io --> to much load *)
    SubscribeFail : BOOL;  (* error if subscribtion on broker fails or if topic isn't valid *)
    TopicValid : TOPIC_VALID;  (* here you get your topic check *)
  END_VAR
  VAR
    SubscribeRising : R_TRIG;
    SubscribeFalling : F_TRIG;
    NeedSubscribe : BOOL;
    NeedUnsubscribe : BOOL;
    SubscribeWasSended : BOOL;
    UnsubscribeWasSended : BOOL;
    MyOutData : DATA_TO_BROKER;
    TimeToResponse : CAA.TICK;
    LastSend : CAA.TICK;
    SendTimeOutTime : ton;
    RecivedQoS : QoS;
    MySplitTopic : HandleSplitTopic;
    RecivedPublishs : ULINT;  (* recived publishs *)
    init : BOOL := FALSE;
    iu : UINT;
  END_VAR

            SUPER^();
//if not config, then leave, do this after super so we calc correct FB numbers
IF NOT DbPointerIo THEN RETURN; END_IF;
GVL_MQTT.ProgNum := PROG_NUM.Subscribe;
SubscribeFalling(CLK:= Subscribe);
SubscribeRising(CLK:= Subscribe);

IF NOT init THEN
	COM_CONFIG := MQTT_IN_OUT^.COM_CONFIG;
	MySplitTopic.LowInit(TopicsLevelInit:= COM_CONFIG.MaxTopicLevels, SplitElementSizeInit:= COM_CONFIG.MaxTopicElementSize, dynMemUsageInit:= ADR(MQTT_IN_OUT^.dynMemUsage));
	init:= TRUE;
END_IF

IF NOT MQTT_IN_OUT^.BROKER_CONNECTED AND SubscribeDone AND Subscribe THEN
	//reconnect after disconnect
	NeedSubscribe := TRUE;
	SubscribeDone := FALSE;
	SubscribeWasSended := FALSE;
	UnsubscribeWasSended := FALSE;
END_IF

IF SubscribeRising.Q THEN
	NeedSubscribe := TRUE;
END_IF


IF SubscribeFalling.Q THEN
	NeedUnsubscribe := TRUE;
END_IF


{info 'reconnect or wait or or or or ....'}
//have to unsubscribe if callback wasn't registered
IF MyOutData.PaketData.CallbackError THEN
	NeedUnsubscribe := TRUE;
	SubscribeFail := TRUE;
END_IF

IF NeedSubscribe AND NOT SubscribeWasSended AND MQTT_IN_OUT^.InFree(* AND CheckToken()*) AND MQTT_IN_OUT^.BROKER_CONNECTED THEN
 
	TopicValid := MySplitTopic.NewTopic(in:= Topic, test:= TRUE, SizeOfString:= 0); //CheckTopicValid(Target:= ADR(SplitTopic)); 
	IF TopicValid = TOPIC_VALID.TOPIC_VALID THEN
		//try to subscribe
		SubscribeWasSended := TRUE;
		//send free
		MQTT_IN_OUT^.IN := ADR(MyOutData);
		MQTT_IN_OUT^.InFree := FALSE;
		MyOutData.PaketData.FbId := MQTT_IN_OUT^.FB_NO_AUTO;
		MyOutData.PaketData.MessageType := MESSAGETYPE.SUBSCRIBE;
		MyOutData.PaketData.MessageQoS := QoSSubscribe;
		MyOutData.PaketData.Callback := Callback;
		MyOutData.PaketData.MqttTopic := Topic;
		MyOutData.PaketData.MqttTopicLength := CommonTypesAndFunctions.LEN(Topic);
		MyOutData.PaketData.SplitTopic := ADR(MySplitTopic);
		MyOutData.PaketData.ExpectingString := ExpectingString;
	
		SubscribeFail := FALSE;
	ELSE
		NeedSubscribe := FALSE;
		SubscribeFail := TRUE;
	END_IF
	ReleaseToken();
END_IF

IF NeedUnsubscribe AND NOT UnsubscribeWasSended AND MQTT_IN_OUT^.InFree(* AND CheckToken() *)AND MQTT_IN_OUT^.BROKER_CONNECTED THEN
	//try to unsubscribe
	UnsubscribeWasSended := TRUE;
	//send free
	MQTT_IN_OUT^.IN := ADR(MyOutData);
	MQTT_IN_OUT^.InFree := FALSE;
	MyOutData.PaketData.FbId := MQTT_IN_OUT^.FB_NO_AUTO;
	MyOutData.PaketData.MessageType := MESSAGETYPE.UNSUBSCRIBE;
	MyOutData.PaketData.MqttTopic := Topic;
	MyOutData.PaketData.MqttTopicLength := CommonTypesAndFunctions.LEN(Topic);
	ReleaseToken();
END_IF

//place behinde send, so leave "Token" to rest....
//here for Subscribe
IF MyOutData.PaketData.SendSucsess AND MyOutData.PaketData.MessageType = MESSAGETYPE.SUBSCRIBE THEN //scusses set by HANDLE_MQTT
	MyOutData.PaketData.SendSucsess := FALSE;
	//paket away...
	SubscribeWasSended := FALSE;
	NeedSubscribe := FALSE; 
	SubscribeDone := TRUE;
	TimeToResponse := TICKS.GetTick(xDummy:= TRUE) - LastSend;
	RecivedQoS := MyOutData.PaketData.SubackQoS;
	IF RecivedQoS = QoS.Fail THEN
		SubscribeFail := TRUE;
	ELSE
		SubscribeFail := FALSE;	
	END_IF
	
END_IF

//here for Unubscribe
IF MyOutData.PaketData.SendSucsess AND MyOutData.PaketData.MessageType = MESSAGETYPE.UNSUBSCRIBE THEN //scusses set by HANDLE_MQTT
	MyOutData.PaketData.SendSucsess := FALSE;
	//paket away...
	UnsubscribeWasSended := FALSE;
	NeedUnsubscribe := FALSE; 
	SubscribeDone := FALSE;
	TimeToResponse := TICKS.GetTick(xDummy:= TRUE) - LastSend;
END_IF

SendTimeOutTime(IN:= NeedSubscribe OR NeedUnsubscribe, PT:= MyConstants.SENDING_TIMEOUT);
SendTimeout := SendTimeOutTime.Q;

          
END_FUNCTION_BLOCK

FUNCTION_BLOCK MQTTValue
  VAR
    Topic : POINTER TO STRING;
    ValueName : POINTER TO STRING;
    ValuePointer : CommonTypesAndFunctions.ALL_TYPES_UNION_POINTER;
    ValueType : CommonTypesAndFunctions.VAR_TYPES;
    ValueDiff : UINT;
    Value : CommonTypesAndFunctions.ALL_TYPES_UNION;
    InitDone : BOOL;
    Send : BOOL;
    SendDone : BOOL;
    OldValue : CommonTypesAndFunctions.ALL_TYPES_UNION;
    RequestToSend : BOOL;
    publish : MQTTPublish;
    PayloadTemplate : STRING(255);
    Payload : STRING(255);
    DecimalPlace : INT;
    ValueString : STRING;
    QoS : QoS;
    RetainMqtt : BOOL;
    PowerForReal : UINT;
    MinTime : TIME;
    MinTimeTimer : ton;
    SendBlock : BOOL;  (* Start block time of sending *)
  END_VAR

            //need to call publish here because of FB nums
publish(
	Topic:= Topic, 
	PayloadString:= ADR(Payload), 
	PublishAsString:= TRUE, 
	QoSIn:= QoS, 
	MRetain:= RetainMqtt, 
	send:= Send, 
	done=> SendDone);

IF NOT InitDone THEN RETURN; END_IF
MinTimeTimer(IN:= SendBlock, PT:= MinTime);
IF MinTimeTimer.Q THEN
	SendBlock := FALSE;
END_IF

Value := CommonTypesAndFunctions.GetValueFromPointer(PointerToValue:= ValuePointer, TypeOfValue:= ValueType);
IF NOT SendBlock THEN
	IF CommonTypesAndFunctions.CheckDeltaValue(Value:= Value,
			 TypeOfValue:= ValueType, DeltaVar:= ValueDiff, LastValue:= OldValue,Faktor:= PowerForReal)THEN
		RequestToSend := TRUE;
	END_IF
END_IF
		 
IF RequestToSend AND NOT Send AND NOT SendBlock THEN
	Payload := PayloadTemplate;
	ValueString := CommonTypesAndFunctions.GetValueString(VALUE:= Value, TypeOfValue:= ValueType, DecimalPlace:= DecimalPlace);
	CommonTypesAndFunctions.concat(s1:= ADR(Payload), s2:= ADR(ValueString));
	Send := TRUE;
	RequestToSend := FALSE;
END_IF

IF SendDone THEN
	Send := FALSE;
	SendBlock := TRUE;
END_IF
          

METHOD Init
  VAR_INPUT
    Topic : POINTER TO STRING;  (* topic name *)
    ValueName : POINTER TO STRING;  (* valuve name, placed with ':' bevor value *)
    ValuePointer : CommonTypesAndFunctions.ALL_TYPES_UNION_POINTER;  (* pointer to value, can be every datatype *)
    ValueType : CommonTypesAndFunctions.VAR_TYPES;  (* type of the var pointet by ValuePointer *)
    ValueDiff : UINT;  (* differenz wich the value have to change bovor it is beeing send. if floting point values it depends on decimals(differen :=1, decimal := 1 --> 0.1 differenz ) *)
    MQTT_IN_OUT : POINTER TO MQTT_IN_OUT;  (* Pointer MQTTT exchange strucure *)
    DecimalPlace : INT;  (* decimal places behind comma on floting point values *)
    QoS : QoS;  (* QoS level of publish *)
    RetainMqtt : BOOL;  (* message should be ratained? *)
    MinTime : TIME;  (* min Time between publish *)
  END_VAR
                  publish.SetMqttInOut(MQTT_IN_OUT := MQTT_IN_OUT);
THIS^.ValuePointer := ValuePointer;
IF ValueDiff = 0 THEN
	THIS^.ValueDiff := 1;
ELSE
	THIS^.ValueDiff := ValueDiff;	
END_IF

THIS^.Topic := Topic;
THIS^.ValueName := ValueName;
THIS^.ValueType := ValueType;
THIS^.PayloadTemplate := ValueName^;
//don't ad ':' if no name is given
IF NOT THIS^.PayloadTemplate[0] = 0 THEN
	CommonTypesAndFunctions.concat(s1:= ADR(THIS^.PayloadTemplate), s2:= ADR(':'));
END_IF
THIS^.DecimalPlace := DecimalPlace;
InitDone := TRUE;
THIS^.RetainMqtt := RetainMqtt;
THIS^.QoS := QoS;
IF THIS^.ValueType = CommonTypesAndFunctions.VAR_TYPES.LREAL_T OR 
	THIS^.ValueType = CommonTypesAndFunctions.VAR_TYPES.REAL_T THEN
	PowerForReal := TO_UINT(EXPT(10,DecimalPlace));
END_IF
THIS^.MinTime := MinTime;
                
END_METHOD
END_FUNCTION_BLOCK

FUNCTION_BLOCK HighLoadPublish
  VAR_INPUT
    ClientID : STRING(255) := 'TestHighRecive/Topic';
    Topic : POINTER TO POINTER TO STRING;
    TopicFix : BOOL;
    payload : POINTER TO POINTER TO STRING;
    PayloadFix : BOOL;
    CountArray : UINT;
    UsedPublishFbs : UINT;
    working : BOOL;  (* set to high to work, low to stop.... *)
    broker : STRING(255);
    QoS : QoS;
    RetainIn : BOOL;
  END_VAR
  VAR_OUTPUT
    finished : BOOL;
  END_VAR
  VAR
    i : UINT;
    Publishs : ARRAY[0..MyConstants.QoS_BUFFER_SIZE] OF MQTTPublish;
    PublishSendBools : ARRAY[0..MyConstants.QoS_BUFFER_SIZE] OF BOOL;
    PublishSendFree : ARRAY[0..MyConstants.QoS_BUFFER_SIZE] OF BOOL := [MyConstants.QoS_BUFFER_SIZE(TRUE)];
    PublishTopicStore : ARRAY[0..MyConstants.QoS_BUFFER_SIZE] OF POINTER TO STRING;
    PublishPayloadStore : ARRAY[0..MyConstants.QoS_BUFFER_SIZE] OF POINTER TO STRING;
    MQTT : HANDLE_MQTT;
    MQTT_INFO : MQTT_INFO;
    init : BOOL;
    MQTT_IN_OUT : MQTT_IN_OUT;
    LastPublished : UINT;
    start : R_TRIG;
    doPublish : BOOL;
  END_VAR

            IF NOT init THEN
	init := TRUE;
	MQTT_IN_OUT.ClientID := ClientID; 
	FOR i := 0 TO UsedPublishFbs - 1 DO
		Publishs[i].SetMqttInOut(MQTT_IN_OUT := ADR(MQTT_IN_OUT));
	END_FOR
END_IF

doPublish := working AND MQTT_INFO.MQTT_CONNECTED;

IF NOT doPublish THEN
	LastPublished := 0;
	FOR i := 0 TO UsedPublishFbs - 1 DO
		PublishSendBools[i] := FALSE;
		Publishs[i](
	send:= PublishSendBools[i]);
	PublishSendFree[i] := TRUE;
	END_FOR
	
END_IF

MQTT(
	MQTT_INFO:= MQTT_INFO, 
	MQTT_IN_OUT:= MQTT_IN_OUT, 
	ENABLE:= TRUE, 
	URL:= broker, 
	TIMEOUT:= T#5S, 
	TLS:= FALSE);
start(CLK := working);

IF start.Q THEN
	finished := FALSE;

END_IF
IF doPublish THEN

	FOR i := 0 TO UsedPublishFbs - 1 DO
		
		IF PublishSendFree[i] AND NOT finished THEN
			PublishSendFree[i] := FALSE;
			
			//get next element
			IF LastPublished >= CountArray THEN
				finished := TRUE;
	
			ELSE
				IF TopicFix THEN
					PublishTopicStore[i] := Topic;
				ELSE
					PublishTopicStore[i] := Topic[LastPublished];	
				END_IF
				
				IF PayloadFix THEN
					PublishPayloadStore[i] := Payload;
				ELSE
					PublishPayloadStore[i] := Payload[LastPublished];	
				END_IF
				
				PublishSendBools[i] := TRUE;
			END_IF
			LastPublished := LastPublished + 1;
			
		END_IF	
		
			Publishs[i](
		Topic:=PublishTopicStore[i], 
		PayloadString:= PublishPayloadStore[i], 
		PublishAsString:= TRUE, 
		QoSIn:= QoS, 
		MRetain:= RetainIn, 
		send:= PublishSendBools[i]);
		IF Publishs[i].done THEN 
			PublishSendFree[i] := TRUE;
		END_IF
		IF Publishs[i].sendActive THEN
			PublishSendBools[i] := FALSE;
		END_IF
	END_FOR
	
END_IF
          
END_FUNCTION_BLOCK

PROGRAM PLC_PRG
  VAR
    MQTT : HANDLE_MQTT;
    MQTT_INFO : MQTT_INFO;
    MQTT_IN_OUT : MQTT_IN_OUT;
    ERROR_C : DWORD;
    ERROR_T : BYTE;
    testPiublish : ARRAY[0..100] OF MQTTPublish;  (* testPiublish: SD_MQTT.MQTTPublish; *)
    init : BOOL := FALSE;
    sendTest : BOOL;
    testtime : ton;
    i : UINT;
    qos : QoS := 2;
    sub1 : MQTTSubscribe;
    con : BOOL;
    recived : BOOL;  (* Testtopic:SD_MQTT.TestcaseCheckTopivValid; TestSubscribe:SD_MQTT.TestSubscribe; *)
    CountSucsess : ARRAY[0..100] OF ULINT;
    MQTTretain : BOOL := TRUE;
    enable : BOOL;
    ReciveData : ARRAY[0..100] OF RECIVE_PAKET;
    reciveIndex : INT;
  END_VAR

            MQTT_IN_OUT.ClientID :='testCodesys';
//MQTT_IN_OUT.PORT := 1883;
//MQTT_IN_OUT.URL := 'test.mosquitto.org';
(*
testtime(IN:= NOT testtime.Q AND sendTest, PT:= T#100MS);
//testtime(IN:= NOT testtime.Q AND sendTest, PT:= T#10S);
IF NOT init THEN
	init := TRUE;
	testPiublish[0].SetMqttInOut(MQTT_IN_OUT := ADR(MQTT_IN_OUT));
	testPiublish[1].SetMqttInOut(MQTT_IN_OUT := ADR(MQTT_IN_OUT));
	testPiublish[2].SetMqttInOut(MQTT_IN_OUT := ADR(MQTT_IN_OUT));
	testPiublish[3].SetMqttInOut(MQTT_IN_OUT := ADR(MQTT_IN_OUT));
	testPiublish[4].SetMqttInOut(MQTT_IN_OUT := ADR(MQTT_IN_OUT));
	testPiublish[5].SetMqttInOut(MQTT_IN_OUT := ADR(MQTT_IN_OUT));
	testPiublish[6].SetMqttInOut(MQTT_IN_OUT := ADR(MQTT_IN_OUT));
	testPiublish[7].SetMqttInOut(MQTT_IN_OUT := ADR(MQTT_IN_OUT));
	testPiublish[8].SetMqttInOut(MQTT_IN_OUT := ADR(MQTT_IN_OUT));
	testPiublish[9].SetMqttInOut(MQTT_IN_OUT := ADR(MQTT_IN_OUT));
	testPiublish[10].SetMqttInOut(MQTT_IN_OUT := ADR(MQTT_IN_OUT));
	testPiublish[11].SetMqttInOut(MQTT_IN_OUT := ADR(MQTT_IN_OUT));
	testPiublish[12].SetMqttInOut(MQTT_IN_OUT := ADR(MQTT_IN_OUT));
	testPiublish[13].SetMqttInOut(MQTT_IN_OUT := ADR(MQTT_IN_OUT));
	testPiublish[14].SetMqttInOut(MQTT_IN_OUT := ADR(MQTT_IN_OUT));
	testPiublish[15].SetMqttInOut(MQTT_IN_OUT := ADR(MQTT_IN_OUT));
	sub1.SetMqttInOut(MQTT_IN_OUT:= ADR(MQTT_IN_OUT));
	//Testtopic();

END_IF

FOR i := 0 TO 20 DO
	CountSucsess[i] := testPiublish[i].CountSend;
END_FOR

//	TestSubscribe();
sub1(
	Subscribe:= con, 
	Topic:= 'test/#', 
	QoSSubscribe:= 2 ,
	Recived => recived
	 );
IF recived THEN
	i:=i;
	ReciveData[reciveIndex].MqttPayload := sub1.PayloadString^;
	ReciveData[reciveIndex].MqttTopic := sub1.TopicOut^;
	reciveIndex := reciveIndex + 1;
	IF reciveIndex > 100 THEN
		reciveIndex := 0;
	END_IF
END_IF
testPiublish[0](
	Topic:= 'test/topic veryyyyyyyyyyyyyyyyyyyyyyyyyyyyyyyyyyyyyyyyyyyyyyyyyyyyyyyyyyyyyyyyyyyyyyyyyyyyyyyyyyyyyyyyyyyyyyyyyyyyyyyyyyyyyyyyyy big topic/1', 
	PayloadString:= 'test pi1', 
	QoSIn:= qos, 
	MRetain:= MQTTretain, 
	send := testtime.Q,
	PublishString := TRUE 
	);
	
testPiublish[1](
	Topic:= 'test/topic veryyyyyyyyyyyyyyyyyyyyyyyyyyyyyyyyyyyyyyyyyyyyyyyyyyyyyyyyyyyyyyyyyyyyyyyyyyyyyyyyyyyyyyyyyyyyyyyyyyyyyyyyyyyyyyyyyy big topic/2', 
	PayloadString:= 'test pi2', 
	QoSIn:= qos, 
	MRetain:= MQTTretain, 
	send := testtime.Q,
	PublishString := TRUE 
	);
testPiublish[2](
	Topic:= 'test/topic veryyyyyyyyyyyyyyyyyyyyyyyyyyyyyyyyyyyyyyyyyyyyyyyyyyyyyyyyyyyyyyyyyyyyyyyyyyyyyyyyyyyyyyyyyyyyyyyyyyyyyyyyyyyyyyyyyy big topic/3', 
	PayloadString:= 'test pi3', 
	QoSIn:= qos, 
	MRetain:= MQTTretain, 
	send := testtime.Q,
	PublishString := TRUE 
	);
testPiublish[3](
	Topic:= 'test/topic veryyyyyyyyyyyyyyyyyyyyyyyyyyyyyyyyyyyyyyyyyyyyyyyyyyyyyyyyyyyyyyyyyyyyyyyyyyyyyyyyyyyyyyyyyyyyyyyyyyyyyyyyyyyyyyyyyy big topic/4', 
	PayloadString:= 'test pi4', 
	QoSIn:= qos, 
	MRetain:= MQTTretain, 
	send := testtime.Q, 
	PublishString := TRUE
	);
testPiublish[4](
	Topic:= 'test/topic veryyyyyyyyyyyyyyyyyyyyyyyyyyyyyyyyyyyyyyyyyyyyyyyyyyyyyyyyyyyyyyyyyyyyyyyyyyyyyyyyyyyyyyyyyyyyyyyyyyyyyyyyyyyyyyyyyy big topic/5', 
	PayloadString:= 'test pi5', 
	QoSIn:= qos, 
	MRetain:= MQTTretain, 
	send := testtime.Q, 
	PublishString := TRUE
	);
testPiublish[5](
	Topic:= 'test/topic veryyyyyyyyyyyyyyyyyyyyyyyyyyyyyyyyyyyyyyyyyyyyyyyyyyyyyyyyyyyyyyyyyyyyyyyyyyyyyyyyyyyyyyyyyyyyyyyyyyyyyyyyyyyyyyyyyy big topic/6', 
	PayloadString:= 'test pi6', 
	QoSIn:= qos, 
	MRetain:= MQTTretain, 
	send := testtime.Q, 
	PublishString := TRUE
	);
testPiublish[6](
	Topic:= 'test/topic veryyyyyyyyyyyyyyyyyyyyyyyyyyyyyyyyyyyyyyyyyyyyyyyyyyyyyyyyyyyyyyyyyyyyyyyyyyyyyyyyyyyyyyyyyyyyyyyyyyyyyyyyyyyyyyyyyy big topic/7', 
	PayloadString:= 'test pi7', 
	QoSIn:= qos, 
	MRetain:= MQTTretain, 
	send := testtime.Q, 
	PublishString := TRUE
	);
testPiublish[7](
	Topic:= 'test/topic veryyyyyyyyyyyyyyyyyyyyyyyyyyyyyyyyyyyyyyyyyyyyyyyyyyyyyyyyyyyyyyyyyyyyyyyyyyyyyyyyyyyyyyyyyyyyyyyyyyyyyyyyyyyyyyyyyy big topic/8', 
	PayloadString:= 'test pi8', 
	QoSIn:= qos, 
	MRetain:= MQTTretain, 
	send := testtime.Q, 
	PublishString := TRUE
	);
testPiublish[8](
	Topic:= 'test/topic veryyyyyyyyyyyyyyyyyyyyyyyyyyyyyyyyyyyyyyyyyyyyyyyyyyyyyyyyyyyyyyyyyyyyyyyyyyyyyyyyyyyyyyyyyyyyyyyyyyyyyyyyyyyyyyyyyy big topic/9', 
	PayloadString:= 'test pi9', 
	QoSIn:= qos, 
	MRetain:= MQTTretain, 
	send := testtime.Q, 
	PublishString := TRUE
	);
testPiublish[9](
	Topic:= 'test/topic veryyyyyyyyyyyyyyyyyyyyyyyyyyyyyyyyyyyyyyyyyyyyyyyyyyyyyyyyyyyyyyyyyyyyyyyyyyyyyyyyyyyyyyyyyyyyyyyyyyyyyyyyyyyyyyyyyy big topic/10', 
	PayloadString:= 'test pi10', 
	QoSIn:= qos, 
	MRetain:= MQTTretain, 
	send := testtime.Q, 
	PublishString := TRUE
	);
testPiublish[10](
	Topic:= 'test/topic veryyyyyyyyyyyyyyyyyyyyyyyyyyyyyyyyyyyyyyyyyyyyyyyyyyyyyyyyyyyyyyyyyyyyyyyyyyyyyyyyyyyyyyyyyyyyyyyyyyyyyyyyyyyyyyyyyy big topic/11', 
	PayloadString:= 'test pi11', 
	QoSIn:= qos, 
	MRetain:= MQTTretain, 
	send := testtime.Q, 
	PublishString := TRUE
	);
testPiublish[11](
	Topic:= 'test/topic veryyyyyyyyyyyyyyyyyyyyyyyyyyyyyyyyyyyyyyyyyyyyyyyyyyyyyyyyyyyyyyyyyyyyyyyyyyyyyyyyyyyyyyyyyyyyyyyyyyyyyyyyyyyyyyyyyy big topic/12', 
	PayloadString:= 'test pi12', 
	QoSIn:= qos, 
	MRetain:= MQTTretain, 
	send := testtime.Q, 
	PublishString := TRUE
	);
testPiublish[12](
	Topic:= 'test/topic veryyyyyyyyyyyyyyyyyyyyyyyyyyyyyyyyyyyyyyyyyyyyyyyyyyyyyyyyyyyyyyyyyyyyyyyyyyyyyyyyyyyyyyyyyyyyyyyyyyyyyyyyyyyyyyyyyy big topic/13', 
	PayloadString:= 'test pi13', 
	QoSIn:= qos, 
	MRetain:= MQTTretain, 
	send := testtime.Q, 
	PublishString := TRUE
	);
testPiublish[13](
	Topic:= 'test/topic veryyyyyyyyyyyyyyyyyyyyyyyyyyyyyyyyyyyyyyyyyyyyyyyyyyyyyyyyyyyyyyyyyyyyyyyyyyyyyyyyyyyyyyyyyyyyyyyyyyyyyyyyyyyyyyyyyy big topic/14', 
	PayloadString:= 'test pi14', 
	QoSIn:= qos, 
	MRetain:= MQTTretain, 
	send := testtime.Q, 
	PublishString := TRUE
	);
testPiublish[14](
	Topic:= 'test/topic veryyyyyyyyyyyyyyyyyyyyyyyyyyyyyyyyyyyyyyyyyyyyyyyyyyyyyyyyyyyyyyyyyyyyyyyyyyyyyyyyyyyyyyyyyyyyyyyyyyyyyyyyyyyyyyyyyy big topic/15', 
	PayloadString:= 'test pi15', 
	QoSIn:= qos, 
	MRetain:= MQTTretain, 
	send := testtime.Q, 
	PublishString := TRUE
	);
testPiublish[15](
	Topic:= 'test/topic veryyyyyyyyyyyyyyyyyyyyyyyyyyyyyyyyyyyyyyyyyyyyyyyyyyyyyyyyyyyyyyyyyyyyyyyyyyyyyyyyyyyyyyyyyyyyyyyyyyyyyyyyyyyyyyyyyy big topic/16', 
	PayloadString:= 'test pi16', 
	QoSIn:= qos, 
	MRetain:= MQTTretain, 
	send := testtime.Q, 
	PublishString := TRUE
	);



(*
MQTT(
	MQTT_INFO:= MQTT_INFO, 
	MQTT_IN_OUT:= MQTT_IN_OUT, 
	ENABLE:= TRUE, 
	URL:= 'test.mosquitto.org:1883', 
	TIMEOUT:= T#5S, 
	ERROR_C=> ERROR_C, 
	ERROR_T=> ERROR_T);
	*)
	(*
	MQTT(
	MQTT_INFO:= MQTT_INFO, 
	MQTT_IN_OUT:= MQTT_IN_OUT, 
	ENABLE:= enable, 
	URL:= 'localhost:1883', 
	TIMEOUT:= T#5S, 
	ERROR_C=> ERROR_C, 
	ERROR_T=> ERROR_T);
	*)



MQTT(
	MQTT_INFO:= MQTT_INFO, 
	MQTT_IN_OUT:= MQTT_IN_OUT, 
	ENABLE:= TRUE, 
	URL:= 'windows-10-pro:1883', 
	TIMEOUT:= T#5S, 
	ERROR_C=> ERROR_C, 
	ERROR_T=> ERROR_T);
*)
          
END_PROGRAM

FUNCTION_BLOCK exampleForFbs
  VAR
    client : ClientWrapper;  (* the MQTT client *)
    FirstExtReciver : FooBarRecivingFB;  (* some reciving FBs *)
    SecondExtReciver : FooBarRecivingFB;
    ThirdExtReciver : FooBarRecivingFB;
    FourthExtReciver : FooBarRecivingFB;
    ArrayRecive : ARRAY[0..9] OF FooBarRecivingFB;  (* a Array of reciving FBs *)
    stock : CallbackCollector;  (* the collector of the FBs *)
  END_VAR

            


client(
	broker:= 'test.mosquitto.org:1883', 
	connect:= TRUE, 
	tls:= FALSE);

	
          
END_FUNCTION_BLOCK

{attribute 'reflection'}
FUNCTION_BLOCK FooBarRecivingFB IMPLEMENTS MQTT_SUBSCRIBE_CALLBACK
  VAR
    {attribute 'instance-path'}
    {attribute 'noinit'}
    instanceName : STRING(255);  (* this string contains the instance name of the FB *)
    LastTreeName : STRING;  (* here we get the "lowest" element of the name... *)
    splitTopic : BOOL;  (* if set to true we search the instance name in the lowest topic *)
    splitPayload : BOOL;  (* if set to true we search the instance name in Payload separatet by the split char *)
    SplitPayloadChar : BYTE;  (* an this is the split char... *)
    Target : STRING(255);  (* here is the target where we will place the payload contend this can be anything... *)
  END_VAR

            
          

METHOD PublishRecived : BOOL
  VAR_INPUT
    Data : CALLBACK_DATA;  (* Collection of recived Data *)
  END_VAR
  VAR
    StrPt : POINTER TO STRING;
  END_VAR
                  // no we can check if the topic/payload fits to my instance name.... 

//now search the right topic 
IF splitTopic THEN
	
	IF CommonTypesAndFunctions.StrEquals(str1:= Data.TopicOutSplit^.Topics[Data.TopicOutSplit^.ValidFields - 1], str2:= ADR(LastTreeName)) THEN
		Target := Data.PayloadString^;
	END_IF

END_IF

//now look into the payload
IF splitPayload THEN
	
	IF CommonTypesAndFunctions.StrEqualsAtStartWithDelimiter(str1:= ADR(LastTreeName), str2:= Data.PayloadString, delimiter:= SplitPayloadChar) THEN
		//now search split char
		StrPt := Data.PayloadString;
		StrPt := StrPt + TO_DWORD(CommonTypesAndFunctions.find(str1 := StrPt, str2:= ADR(SplitPayloadChar))) + 1;
		Target := StrPt^;
	END_IF
END_IF

                
END_METHOD

METHOD initAsFindTopic : BOOL
                  getLastTreeName();
splitPayload := FALSE;
splitTopic := TRUE;
                
END_METHOD

METHOD getLastTreeName : BOOL
                  LastTreeName := CommonTypesAndFunctions.FindLasDot(ADR(instanceName))^;

                
END_METHOD

METHOD initAsFindPayload : BOOL
  VAR_INPUT
    splitChar : STRING;  (* only first char is selected *)
  END_VAR
                  getLastTreeName();
splitPayload := TRUE;
splitTopic := FALSE;

SplitPayloadChar := CommonTypesAndFunctions.GetChar(in:= splitChar);
                
END_METHOD
END_FUNCTION_BLOCK

FUNCTION_BLOCK TestcaseCheckTopivValid
  VAR
    t1 : HandleSplitTopic;
    s100 : STRING(101) := '1111111111111111111111111111111111111111111111111111111111111111111111111111111111111111111111111111';
    splus : STRING := '+';
    ssharp : STRING := '#';
    stest : STRING := 'test';
    valids : ARRAY[0..30] OF STRING := ['/+//sdf/test1', '/sd//', 'test1/+/rest/#', 'test1/#', 'test1/topic2/+/Topic3/+/5636/ggesd', '///', '///+//sdf/test1//', '//+//sdf/test1/', '#', '', '', '', '', '', ''];
    falses : ARRAY[0..30] OF STRING := ['test1/topic2/+/Topic3#/', 'test1/#/topic2/+/Topic3/#456', 'test1+', 'test1/#/topic2/+/Topic3/+/5636/ggesd', 'test1#', '', '', '', '', '', '', '', '', '', ''];
    s1 : STRING(64000);
    valid : TOPIC_VALID;
    pts : ARRAY[0..20] OF POINTER TO STRING;
    sp : POINTER TO SPLIT_TOPIC;
    COM_CONFIG : COM_CONFIG;
    dynMemUsage : UDINT;
  END_VAR

            	(*GetSplitTopic(in:= 'test1/topic2/+/Topic3#/', Target:= ADR(dis1), CountSplitTopicSizeExceeded:= ADR(CountSplitTopicSizeExceeded));
	
	GetSplitTopic(in:= 'test1/#/topic2/+/Topic3/#456', Target:= ADR(dis2), CountSplitTopicSizeExceeded:= ADR(CountSplitTopicSizeExceeded));
	GetSplitTopic(in:= 'test1/+/rest/#', Target:= ADR(dis3), CountSplitTopicSizeExceeded:= ADR(CountSplitTopicSizeExceeded));
	GetSplitTopic(in:= 'test1/#', Target:= ADR(dis4), CountSplitTopicSizeExceeded:= ADR(CountSplitTopicSizeExceeded));
	GetSplitTopic(in:= 'test1/topic2/+/Topic3/+/5636/ggesd', Target:= ADR(dis5), CountSplitTopicSizeExceeded:= ADR(CountSplitTopicSizeExceeded));
	GetSplitTopic(in:= 'test1/#/topic2/+/Topic3/+/5636/ggesd', Target:= ADR(dis6), CountSplitTopicSizeExceeded:= ADR(CountSplitTopicSizeExceeded));
	GetSplitTopic(in:= 'test1#', Target:= ADR(dis7), CountSplitTopicSizeExceeded:= ADR(CountSplitTopicSizeExceeded));
	GetSplitTopic(in:= 'test1+', Target:= ADR(dis8), CountSplitTopicSizeExceeded:= ADR(CountSplitTopicSizeExceeded));
	GetSplitTopic(in:= '/+//sdf/test1', Target:= ADR(dis9), CountSplitTopicSizeExceeded:= ADR(CountSplitTopicSizeExceeded));
	GetSplitTopic(in:= '//+//sdf/test1/', Target:= ADR(dis10), CountSplitTopicSizeExceeded:= ADR(CountSplitTopicSizeExceeded));
	GetSplitTopic(in:= '///+//sdf/test1//', Target:= ADR(dis11), CountSplitTopicSizeExceeded:= ADR(CountSplitTopicSizeExceeded));
	GetSplitTopic(in:= '///', Target:= ADR(dis12), CountSplitTopicSizeExceeded:= ADR(CountSplitTopicSizeExceeded));
	GetSplitTopic(in:= '/sd//', Target:= ADR(dis13), CountSplitTopicSizeExceeded:= ADR(CountSplitTopicSizeExceeded));
	Valid1:=CheckTopicValid(Target:= ADR(dis1));
	Valid2:=CheckTopicValid(Target:= ADR(dis2));
	Valid3:=CheckTopicValid(Target:= ADR(dis3));
	Valid4:=CheckTopicValid(Target:= ADR(dis4));
	Valid5:=CheckTopicValid(Target:= ADR(dis5));
	Valid6:=CheckTopicValid(Target:= ADR(dis6));
	Valid7:=CheckTopicValid(Target:= ADR(dis7));
	Valid8:=CheckTopicValid(Target:= ADR(dis8));
	Valid9:=CheckTopicValid(Target:= ADR(dis9));
	*)
	
	t1.LowInit(SplitElementSizeInit:=400, TopicsLevelInit:= 40, dynMemUsageInit:= ADR(dynMemUsage));
	valid := t1.NewTopic(in := ADR(valids[0]), test:= TRUE, SizeOfString:= 0);
	sp := t1.GetSplitTopic();
	pts[0] := sp^.Topics[0];
	pts[1] := sp^.Topics[1];
	pts[2] := sp^.Topics[2];
	pts[3] := sp^.Topics[3];
	pts[4] := sp^.Topics[4];
	pts[5] := sp^.Topics[5];
	pts[6] := sp^.Topics[6];
	pts[7] := sp^.Topics[7];
	pts[8] := sp^.Topics[8];
	valid := t1.NewTopic(in := ADR(valids[1]), test:= TRUE, SizeOfString:= 0);
	valid := t1.NewTopic(in := ADR(valids[2]), test:= TRUE, SizeOfString:= 0);
	valid := t1.NewTopic(in := ADR(valids[3]), test:= TRUE, SizeOfString:= 0);
	valid := t1.NewTopic(in := ADR(valids[4]), test:= TRUE, SizeOfString:= 0);
	valid := t1.NewTopic(in := ADR(valids[5]), test:= TRUE, SizeOfString:= 0);
	valid := t1.NewTopic(in := ADR(valids[6]), test:= TRUE, SizeOfString:= 0);
	valid := t1.NewTopic(in := ADR(valids[7]), test:= TRUE, SizeOfString:= 0);
	valid := t1.NewTopic(in := ADR(valids[8]), test:= TRUE, SizeOfString:= 0);
	
	valid := t1.NewTopic(in := ADR(falses[0]), test:= TRUE, SizeOfString:= 0);
	valid := t1.NewTopic(in := ADR(falses[1]), test:= TRUE, SizeOfString:= 0);
	valid := t1.NewTopic(in := ADR(falses[2]), test:= TRUE, SizeOfString:= 0);
	valid := t1.NewTopic(in := ADR(falses[3]), test:= TRUE, SizeOfString:= 0);
	valid := t1.NewTopic(in := ADR(falses[4]), test:= TRUE, SizeOfString:= 0);
	valid := t1.NewTopic(in := ADR(falses[5]), test:= TRUE, SizeOfString:= 0);
	valid := t1.NewTopic(in := ADR(falses[6]), test:= TRUE, SizeOfString:= 0);
	valid := t1.NewTopic(in := ADR(falses[7]), test:= TRUE, SizeOfString:= 0);
	
	
	//now bulid some realy big topics and thest them....
	s1 :='';
	CommonTypesAndFunctions.concat(s1:= ADR(s1), s2:= ADR('/'));
	CommonTypesAndFunctions.concat(s1:= ADR(s1), s2:= ADR(s100));
	CommonTypesAndFunctions.concat(s1:= ADR(s1), s2:= ADR('/'));
	CommonTypesAndFunctions.concat(s1:= ADR(s1), s2:= ADR(splus));
	CommonTypesAndFunctions.concat(s1:= ADR(s1), s2:= ADR('/'));
	CommonTypesAndFunctions.concat(s1:= ADR(s1), s2:= ADR(s100));
	CommonTypesAndFunctions.concat(s1:= ADR(s1), s2:= ADR('/'));
	CommonTypesAndFunctions.concat(s1:= ADR(s1), s2:= ADR(s100));
	CommonTypesAndFunctions.concat(s1:= ADR(s1), s2:= ADR('/'));
	CommonTypesAndFunctions.concat(s1:= ADR(s1), s2:= ADR(ssharp));
	//valid
	valid := t1.NewTopic(in := ADR(s1), test:= TRUE, SizeOfString:= 0);
	s1 :='';
	CommonTypesAndFunctions.concat(s1:= ADR(s1), s2:= ADR('/'));
	CommonTypesAndFunctions.concat(s1:= ADR(s1), s2:= ADR(s100));
	CommonTypesAndFunctions.concat(s1:= ADR(s1), s2:= ADR('/'));
	CommonTypesAndFunctions.concat(s1:= ADR(s1), s2:= ADR(splus));
	CommonTypesAndFunctions.concat(s1:= ADR(s1), s2:= ADR('/'));
	CommonTypesAndFunctions.concat(s1:= ADR(s1), s2:= ADR(s100));
	CommonTypesAndFunctions.concat(s1:= ADR(s1), s2:= ADR('/'));
	CommonTypesAndFunctions.concat(s1:= ADR(s1), s2:= ADR(s100));
	CommonTypesAndFunctions.concat(s1:= ADR(s1), s2:= ADR('/'));
	CommonTypesAndFunctions.concat(s1:= ADR(s1), s2:= ADR(ssharp));
	CommonTypesAndFunctions.concat(s1:= ADR(s1), s2:= ADR('/'));
	//not valid # not at last pos
	valid := t1.NewTopic(in := ADR(s1), test:= TRUE, SizeOfString:= 0);
	s1 :='';
	CommonTypesAndFunctions.concat(s1:= ADR(s1), s2:= ADR('/'));
	CommonTypesAndFunctions.concat(s1:= ADR(s1), s2:= ADR(s100));
	CommonTypesAndFunctions.concat(s1:= ADR(s1), s2:= ADR('/'));
	CommonTypesAndFunctions.concat(s1:= ADR(s1), s2:= ADR(splus));
	CommonTypesAndFunctions.concat(s1:= ADR(s1), s2:= ADR('/'));
	CommonTypesAndFunctions.concat(s1:= ADR(s1), s2:= ADR(s100));
	CommonTypesAndFunctions.concat(s1:= ADR(s1), s2:= ADR(splus));
	CommonTypesAndFunctions.concat(s1:= ADR(s1), s2:= ADR('/'));
	CommonTypesAndFunctions.concat(s1:= ADR(s1), s2:= ADR(s100));
	CommonTypesAndFunctions.concat(s1:= ADR(s1), s2:= ADR('/'));
	CommonTypesAndFunctions.concat(s1:= ADR(s1), s2:= ADR(ssharp));
	
	//not valid + within topic
	valid := t1.NewTopic(in := ADR(s1), test:= TRUE, SizeOfString:= 0);
	
	s1 :='';
	CommonTypesAndFunctions.concat(s1:= ADR(s1), s2:= ADR('/'));
	CommonTypesAndFunctions.concat(s1:= ADR(s1), s2:= ADR(s100));
	CommonTypesAndFunctions.concat(s1:= ADR(s1), s2:= ADR('/'));
	CommonTypesAndFunctions.concat(s1:= ADR(s1), s2:= ADR(splus));
	CommonTypesAndFunctions.concat(s1:= ADR(s1), s2:= ADR('/'));
	CommonTypesAndFunctions.concat(s1:= ADR(s1), s2:= ADR(s100));
	CommonTypesAndFunctions.concat(s1:= ADR(s1), s2:= ADR(ssharp));
	CommonTypesAndFunctions.concat(s1:= ADR(s1), s2:= ADR('/'));
	CommonTypesAndFunctions.concat(s1:= ADR(s1), s2:= ADR(s100));
	CommonTypesAndFunctions.concat(s1:= ADR(s1), s2:= ADR('/'));
	CommonTypesAndFunctions.concat(s1:= ADR(s1), s2:= ADR(ssharp));
	
	//not valid # within topic
	valid := t1.NewTopic(in := ADR(s1), test:= TRUE, SizeOfString:= 0);
          
END_FUNCTION_BLOCK

FUNCTION_BLOCK testHighLoadPublish
  VAR_INPUT
    topics : UINT := TEST_TOPICS;
    broker : STRING := 'test.mosquitto.org:1883';
    addTopic : STRING(200);
    retpeatTime : TIME := TIME#1m0s0ms;
  END_VAR
  VAR
    HighLoad : HighLoadPublish;
    init : BOOL;
    i : UINT;
    testTopic : STRING(255) := 'High Payload Test with very very very very very very very very very very big topic/Outs';  (* testTopics:ARRAY[0..TOPICS_MAX] OF STRING(255); *)
    testPayload : ARRAY[0..TOPICS_MAX] OF STRING(255);
    splitChar : STRING := '=';
    PayloadPrefix : STRING := 'Output:';
    RecivePayloadStore : ARRAY[0..TOPICS_MAX] OF LINT;  (* testPayloadRecive:ARRAY[0..TOPICS_MAX]OF STRING; *)
    SendPayloadStore : ARRAY[0..TOPICS_MAX] OF STRING(255);
    SendPayloadStorePointerArray : ARRAY[0..TOPICS_MAX] OF POINTER TO STRING;
    tmpString : STRING;
    tmpString2 : STRING;
    step : INT;
    nextRun : BOOL;
    tNewRun : ton;
    work : BOOL;
  END_VAR
  VAR CONSTANT
    TEST_TOPICS : UINT := 200;
    TOPICS_MAX : UINT := 10000;
  END_VAR

            IF NOT init THEN
	 init := TRUE;
	//Testtopic();
	FOR i := 0 TO topics - 1 DO
		
		tmpString := PayloadPrefix;
		tmpString2 := UINT_TO_STRING(i);
		CommonTypesAndFunctions.concat(s1:= ADR(tmpString), s2:= ADR(tmpString2));
		
		CommonTypesAndFunctions.concat(s1:= ADR(tmpString), s2:= ADR(splitChar));
		CommonTypesAndFunctions.concat(s1:= ADR(tmpString), s2:= ADR(tmpString2));
		SendPayloadStore[i] := tmpString;
		SendPayloadStorePointerArray[i] := ADR(SendPayloadStore[i]);
		step := 10;
	END_FOR
	
END_IF

HighLoad(
	ClientID:= 'Test for HighLoadPublish', 
	Topic:= ADR(testTopic), 
	TopicFix:= TRUE, 
	payload:= ADR(SendPayloadStorePointerArray[0]),
	PayloadFix := FALSE, 
	CountArray:= topics, 
	UsedPublishFbs:= MyConstants.QoS_BUFFER_SIZE - 1, 
	working:= work, 
	broker:= 'windows-10-pro:1883', 
	QoS:= QoS.ExactlyOnce, 
	RetainIn:= FALSE);

IF topics >= TOPICS_MAX THEN
	topics := TOPICS_MAX - 1;
END_IF


	
CASE step OF
	10: //empty
		step := 20;
	
	20: 
		work := TRUE; 
		step := 30;
	30: //wait for finish
		IF HighLoad.finished THEN
			work := FALSE;
			step := 40;
			
		END_IF
		
	40: //wait for next run
		IF tNewRun.Q OR nextRun THEN
			step := 10;
		END_IF 
END_CASE

tNewRun(in := step = 40,PT:= retpeatTime);
          
END_FUNCTION_BLOCK

FUNCTION_BLOCK testHighRecive
  VAR_INPUT
    topics : UINT := TEST_TOPICS;
    broker : STRING := 'test.mosquitto.org:1883';
    addTopic : STRING(200);
    repeatTime : TIME := TIME#1m0s0ms;
  END_VAR
  VAR
    MQTT : HANDLE_MQTT;
    MQTT_INFO : MQTT_INFO;
    send : HighLoadPublish;  (* pub:MQTTPublish; *)
    sendWork : BOOL;
    PayloadTarget : POINTER TO POINTER TO STRING;
    subs : MQTTSubscribe;
    MQTT_IN_OUT : MQTT_IN_OUT;
    tNewRun : TON;
    init : BOOL;
    i : UINT;
    testPayload : ARRAY[0..TOPICS_MAX] OF STRING;
    testPayloadPointer : ARRAY[0..TOPICS_MAX] OF POINTER TO STRING;
    emptyString : STRING := '';
    pointerToEmptyString : POINTER TO STRING := ADR(emptyString);
    testTopics : ARRAY[0..TOPICS_MAX] OF STRING(255);
    testTopicsPointer : ARRAY[0..TOPICS_MAX] OF POINTER TO STRING;
    compareTopic : ARRAY[0..TOPICS_MAX] OF STRING(255);
    testPayloadRecive : ARRAY[0..TOPICS_MAX] OF STRING;
    PayloadReciveValue : ARRAY[0..TOPICS_MAX] OF STRING(255);
    SplitChar : STRING := '=';
    tmpString : STRING;
    step : INT;
    topic : STRING(255);
    payload : STRING(255);
    sendPublish : BOOL;
    subscribe : BOOL;
    noData : BOOL;
    nextRun : BOOL;
    ListCallback : ListStringCallback;
    CallbackData : ARRAY[0..TOPICS_MAX] OF LIST_STRING_CALLBACK_DATA;
    PayloadFix : BOOL;
  END_VAR
  VAR CONSTANT
    TEST_TOPICS : UINT := 200;
    TOPICS_MAX : UINT := 10000;
  END_VAR

            IF NOT init THEN
	init := TRUE;
	//pub.SetMqttInOut(MQTT_IN_OUT := ADR(MQTT_IN_OUT));
	
	subs.SetMqttInOut(MQTT_IN_OUT:= ADR(MQTT_IN_OUT));
	//Testtopic();
	FOR i := 0 TO topics - 1 DO
		tmpString := UINT_TO_STRING(i);
		testTopics[i] := 'RetainTopicSD/Topic:';
		CommonTypesAndFunctions.concat(s1:= ADR(testTopics[i]), s2:= ADR(addTopic));
		CommonTypesAndFunctions.concat(s1:= ADR(testTopics[i]), s2:= ADR(tmpString));
		testTopicsPointer[i] := ADR(testTopics[i]);
		testPayloadPointer[i] := ADR(testPayload[i]);
		//CommonTypesAndFunctions.concat(s1:= ADR(testTopics[i]), s2:= ADR('/'));
		testPayload[i] := tmpString;
		compareTopic[i] :='Topic:';
		CommonTypesAndFunctions.concat(s1:= ADR(compareTopic[i]), s2:= ADR(addTopic));
		CommonTypesAndFunctions.concat(s1:= ADR(compareTopic[i]), s2:= ADR(tmpString));
		
		//compareTopic[i] := tmpString;
		CallbackData[i].SubTopic := ADR(compareTopic[i]);
		CallbackData[i].Target := ADR(testPayloadRecive[i]);
	END_FOR
	ListCallback.InitAsSplitTopic(ListData:= ADR(CallbackData[0]), LengthOfData:= i);
END_IF
IF topics >= TOPICS_MAX THEN
	topics := TOPICS_MAX;
END_IF

send(
	ClientID:= 'SendHighRecive test', 
	Topic:= ADR(testTopicsPointer), 
	TopicFix:= FALSE, 
	payload:= PayloadTarget, 
	PayloadFix := PayloadFix,
	CountArray:= topics, 
	UsedPublishFbs:= 48, 
	working:= sendWork, 
	broker:= broker, 
	QoS:= QoS.ExactlyOnce, 
	RetainIn:= TRUE);
subs(
	Subscribe:= subscribe, 
	Topic:= ADR('RetainTopicSD/#'), 
	QoSSubscribe:= QoS.ExactlyOnce, 
	ExpectingString:= TRUE,
	Callback := ListCallback);
	

MQTT(
	MQTT_INFO:= MQTT_INFO, 
	MQTT_IN_OUT:= MQTT_IN_OUT, 
	ENABLE:= TRUE, 
	URL:= broker, 
	TIMEOUT:= T#5S, 
	TLS:= FALSE);
IF NOT MQTT_INFO.MQTT_CONNECTED THEN
	step := 0;
END_IF
	
CASE step OF
	0: 	step := 1;
		
		FOR i := 0 TO topics - 1 DO
			testPayloadRecive[i] := '';
		END_FOR
	1: IF MQTT_INFO.MQTT_CONNECTED THEN
			step:= 10;
			PayloadTarget := ADR(testPayloadPointer); 
			sendWork := TRUE;
			PayloadFix := FALSE;
		END_IF
	10: //publish all data
		IF send.finished THEN
			sendWork := FALSE;
			step := 30; 
			
		END_IF
	
	30: subscribe := TRUE;
		step := 40;
		
	40: // wait to recive all topics
		noData := FALSE;
		FOR i := 0 TO topics - 1 DO
			IF testPayloadRecive[i] <> testPayload[i] THEN
				noData := TRUE;
			END_IF
		END_FOR
		IF NOT noData THEN
			step := 50; 
		END_IF 
		//unsubscripe
	50: subscribe := FALSE;
		step := 52;
		PayloadTarget := pointerToEmptyString; 
		//cleanup recive buffer
		FOR i := 0 TO topics - 1 DO
			testPayloadRecive[i] :='';
		END_FOR
		sendWork := TRUE;
		PayloadFix := TRUE;
	52: //discharge retain messages from broker
		IF send.finished  THEN
			sendWork := FALSE;
			step := 60;
		END_IF
	
	60:
		IF nextRun OR tNewRun.Q THEN 
			nextRun := FALSE;
			step := 0;
		END_IF
END_CASE

tNewRun(in := step = 60,PT:= repeatTime);
          
END_FUNCTION_BLOCK

FUNCTION_BLOCK testHighReciveSplitPayload
  VAR_INPUT
    Count : UINT := TEST_TOPICS;
    broker : STRING := 'test.mosquitto.org:1883';
    addTopic : STRING(200);
    repeatTime : TIME := TIME#1m0s0ms;
  END_VAR
  VAR
    MQTT_RECIVE : HANDLE_MQTT;
    MQTT_INFO_RECIVE : MQTT_INFO;
    subs : MQTTSubscribe;
    MQTT_IN_OUT_RECIVE : MQTT_IN_OUT;
    tNewRun : TON;
    init : BOOL;
    i : UINT;
    testTopic : STRING := 'SD_MQTT/TEST_PAYLOAD/PAYLOAD';  (* testTopics:ARRAY[0..TOPICS_MAX] OF STRING(255); *)
    testPayloadString : ARRAY[0..TOPICS_MAX] OF STRING(255);
    splitChar : STRING := '=';
    PayloadPrefix : STRING := 'Output';
    comparePayload : ARRAY[0..TOPICS_MAX] OF STRING(255);
    SendPayloadStorePointerArray : ARRAY[0..TOPICS_MAX] OF POINTER TO STRING;  (* testPayloadRecive:ARRAY[0..TOPICS_MAX]OF STRING; *)
    RecivePayloadStore : ARRAY[0..TOPICS_MAX] OF LINT;
    SendPayloadStore : ARRAY[0..TOPICS_MAX] OF LINT;
    tmpString : STRING;
    tmpString2 : STRING;
    step : UINT;
    subscribe : BOOL;
    HighSendPublish : HighLoadPublish;
    runPublishWorker : BOOL;
    noData : BOOL;
    nextRun : BOOL;
    ListCallback : ListAllValuesCallback;
    CallbackData : ARRAY[0..TOPICS_MAX] OF LIST_ALLVALUES_CALLBACK_DATA;
  END_VAR
  VAR CONSTANT
    TEST_TOPICS : UINT := 200;
    TOPICS_MAX : UINT := 10000;
  END_VAR

            IF NOT init THEN
	init := TRUE;
	MQTT_IN_OUT_RECIVE.ClientID := 'Test Client Recive';
	subs.SetMqttInOut(MQTT_IN_OUT:= ADR(MQTT_IN_OUT_RECIVE));
	//Testtopic();
	FOR i := 0 TO Count - 1 DO

		tmpString := PayloadPrefix;
		tmpString2 := UINT_TO_STRING(i);
		CommonTypesAndFunctions.concat(s1:= ADR(tmpString), s2:= ADR(tmpString2));
		//finished building compare payload
		comparePayload[i] := tmpString;
		CommonTypesAndFunctions.concat(s1:= ADR(tmpString), s2:= ADR(splitChar));
		SendPayloadStore[i] := i + 22;
		tmpString2 := TO_STRING(SendPayloadStore[i]);
		CommonTypesAndFunctions.concat(s1:= ADR(tmpString), s2:= ADR(tmpString2));
		//CommonTypesAndFunctions.concat(s1:= ADR(tmpString), s2:= ADR(splitChar));
		
		testPayloadString[i] := tmpString; 
		
		//compareTopic[i] := tmpString;
		CallbackData[i].SubTopic := ADR(comparePayload[i]);
		CallbackData[i].Target.POINTER_TO_LINT_T := ADR(RecivePayloadStore[i]);
		CallbackData[i].VarTYPE := CommonTypesAndFunctions.VAR_TYPES.LINT_T;
		SendPayloadStorePointerArray[i] := ADR(testPayloadString[i]);
	END_FOR
	ListCallback.InitAsSplitPayload(Data:= ADR(CallbackData[0]), LengthOfData:= i, SplitChar:= CommonTypesAndFunctions.GetChar(splitChar));
END_IF
IF Count >= TOPICS_MAX THEN
	Count := TOPICS_MAX;
END_IF

subs(
	Subscribe:= subscribe, 
	Topic:= ADR(testTopic), 
	QoSSubscribe:= QoS.ExactlyOnce, 
	ExpectingString:= TRUE,
	Callback := ListCallback);
	
MQTT_RECIVE(
	MQTT_INFO:= MQTT_INFO_RECIVE, 
	MQTT_IN_OUT:= MQTT_IN_OUT_RECIVE, 
	ENABLE:= TRUE, 
	URL:= broker, 
	TIMEOUT:= T#5S, 
	TLS:= FALSE);
IF NOT MQTT_INFO_RECIVE.MQTT_CONNECTED THEN
	step := 0;
END_IF
	
HighSendPublish(
	ClientID:= 'HighSendClient', 
	Topic:= ADR(testTopic), 
	TopicFix:= TRUE, 
	payload:= ADR(SendPayloadStorePointerArray), 
	CountArray:= Count, 
	UsedPublishFbs:= 49, 
	working:= runPublishWorker, 
	broker:= broker, 
	QoS:= QoS.ExactlyOnce, 
	RetainIn:= FALSE);


CASE step OF
	0: 	step := 1;
		FOR i := 0 TO Count - 1 DO
			RecivePayloadStore[i] := 0;
		END_FOR
	1: IF MQTT_INFO_RECIVE.MQTT_CONNECTED THEN
			step:= 5;
			//subscribe
			subscribe := TRUE;
		END_IF
	5: //wait for subscribe
		IF subs.SubscribeDone THEN
			step:= 10;
		END_IF
		 
	10: //publish all and recive data
		//start publish
		runPublishWorker := TRUE;
		step := 20;
	20: IF HighSendPublish.finished THEN
		//wait until send is done		
			runPublishWorker := FALSE;
			step:= 30;

		END_IF
	30: //now check payload
		
			noData := FALSE;
		FOR i := 0 TO Count - 1 DO
			IF RecivePayloadStore[i] <> SendPayloadStore[i] THEN
				noData := TRUE;
				EXIT;
			END_IF
		END_FOR
		IF NOT noData THEN
			step := 40;
			//unsubscripe
			subscribe := FALSE; 
		END_IF	
	40: 
		IF nextRun OR tNewRun.Q THEN 
			nextRun := FALSE;
			step := 0;
		END_IF
END_CASE

tNewRun(in := step = 40,PT:= repeatTime);
          
END_FUNCTION_BLOCK

FUNCTION_BLOCK TestLongPublish
  VAR_INPUT
    broker : STRING := 'test.mosquitto.org';
  END_VAR
  VAR
    longPayload : STRING(8000);
    longTopic : STRING(8000) := 'TestTopic/';
    longPayloadRecive : STRING(8000);
    longTopicRecive : STRING(8000);
    init : BOOL;
    i1 : UINT;
    i2 : UINT;
    countAsciis : UINT := 48;
    pt1 : POINTER TO BYTE;
    pt2 : POINTER TO BYTE;
    step : UINT;
    MQTT : HANDLE_MQTT;
    MQTT_INFO : MQTT_INFO;
    MQTT_IN_OUT : MQTT_IN_OUT;
    ComConfig : COM_CONFIG;
    pup : MQTTPublish;
    SUB1 : MQTTSubscribe;
    callback : SingelStringCallback;
    connect : BOOL;
  END_VAR

            IF NOT init THEN
	init := TRUE;
	
	ComConfig.MaxPayloadSize := 20000;
	ComConfig.MaxTopicLevels := 10;
	ComConfig.MaxTopicElementSize := 10000;
	
	MQTT_IN_OUT.ClientID := 'TestCodesys';
	MQTT_IN_OUT.COM_CONFIG := ComConfig;
	//firs build some nice pacload ...
	pt1 := ADR(longPayload);
	pt2 := ADR(longTopic);
	pt2 := pt2 + 10;
	FOR i1 := 0 TO 8000 / countAsciis - 1 DO
		FOR i2 := 0 TO countAsciis DO
			pt1^ := TO_BYTE(i2 + 16#30); //16#30 --> ASCII zero
			pt2^ := TO_BYTE(i2 + 16#30); //16#30 --> ASCII zero
			pt1 := pt1 + 1;
			pt2 := pt2 + 1;
		END_FOR
	END_FOR
	
	callback.Init(payload:= ADR(longPayloadRecive), topic:= ADR(longTopicRecive));
END_IF


MQTT(
	MQTT_INFO:= MQTT_INFO, 
	MQTT_IN_OUT:= MQTT_IN_OUT, 
	ENABLE:= connect, 
	URL:= broker, 
	TIMEOUT:= , 
	TLS:= , 
	ERROR_C=> , 
	ERROR_T=> );


CASE step OF 
	0://begin
		//connect
END_CASE
          
END_FUNCTION_BLOCK

FUNCTION_BLOCK TestMqtt
  VAR_INPUT
    clientID : STRING := 'testCodesys';
  END_VAR
  VAR
    MQTT : HANDLE_MQTT;
    MQTT_INFO : MQTT_INFO;
    MQTT_IN_OUT : MQTT_IN_OUT;
    ERROR_C : DWORD;
    ERROR_T : BYTE;
    testPiublish : ARRAY[0..100] OF MQTTPublish;  (* testPiublish: SD_MQTT.MQTTPublish; *)
    init : BOOL := FALSE;
    sendTest : BOOL;
    testBigPublish : BOOL;
    testBigPayload : BOOL;
    testTimeBigPublish : ton;
    testTimeBigPayload : ton;
    testtime : ton;
    i : UDINT;
    qos : QoS := 2;
    sub1 : MQTTSubscribe;
    sub2 : MQTTSubscribe;
    sub3 : MQTTSubscribe;
    con : BOOL;
    TestLongSubscribe : BOOL;
    recived1 : BOOL;  (* Testtopic:SD_MQTT.TestcaseCheckTopivValid; TestSubscribe:SD_MQTT.TestSubscribe; *)
    recived2 : BOOL;
    recived3 : BOOL;
    longRecived : BOOL;
    CountSucsess : ARRAY[0..100] OF ULINT;
    MQTTretain : BOOL := TRUE;
    enable : BOOL;
    ReciveData : ARRAY[0..100] OF RECIVE_PAKET;
    reciveIndex : INT;
    TestLen : UINT;
    SubscribeForBigPaket : BOOL;
    t1 : HandleSplitTopic;
    s100 : STRING(101) := '1111111111111111111111111111111111111111111111111111111111111111111111111111111111111111111111111111';
    sa : STRING := 'abcdefghijklmnopqrstuvwxyz';
    sb : STRING := 'ABCDEFGHIJKLMNOPQRSTUVWXYZ';
    sc : STRING := '0123456789';
    sd : STRING := '9876543210';
    splus : STRING := '+';
    ssharp : STRING := '#';
    stest : STRING := 'test';
    s1 : STRING(64000);
    s2 : STRING(64000);
    b1 : ARRAY[0..(bSize + 2)] OF BYTE;
  END_VAR
  VAR CONSTANT
    bSize : UDINT := ((1024 * 1024) * 30);
  END_VAR

            MQTT_IN_OUT.ClientID :=clientID;
MQTT_IN_OUT.COM_CONFIG.MaxPayloadSize :=50000;
MQTT_IN_OUT.COM_CONFIG.MaxTopicLevels := 200;
//MQTT_IN_OUT.PORT := 1883;
//MQTT_IN_OUT.URL := 'test.mosquitto.org';


{info 'TODO make some nice test cases'}




//testtime(IN:= , PT:= );
testtime(IN:= NOT testtime.Q AND sendTest, PT:= T#50MS);
testTimeBigPublish(IN:= NOT testTimeBigPublish.Q AND testBigPublish, PT:= T#100MS);
testTimeBigPayload(IN:= NOT testTimeBigPayload.Q AND testBigPayload, PT:= T#100MS);
//testtime(IN:= NOT testtime.Q AND sendTest, PT:= T#10S);
IF NOT init THEN
	init := TRUE;
	testPiublish[0].SetMqttInOut(MQTT_IN_OUT := ADR(MQTT_IN_OUT));
	testPiublish[1].SetMqttInOut(MQTT_IN_OUT := ADR(MQTT_IN_OUT));
	testPiublish[2].SetMqttInOut(MQTT_IN_OUT := ADR(MQTT_IN_OUT));
	testPiublish[3].SetMqttInOut(MQTT_IN_OUT := ADR(MQTT_IN_OUT));
	testPiublish[4].SetMqttInOut(MQTT_IN_OUT := ADR(MQTT_IN_OUT));
	testPiublish[5].SetMqttInOut(MQTT_IN_OUT := ADR(MQTT_IN_OUT));
	testPiublish[6].SetMqttInOut(MQTT_IN_OUT := ADR(MQTT_IN_OUT));
	testPiublish[7].SetMqttInOut(MQTT_IN_OUT := ADR(MQTT_IN_OUT));
	testPiublish[8].SetMqttInOut(MQTT_IN_OUT := ADR(MQTT_IN_OUT));
	testPiublish[9].SetMqttInOut(MQTT_IN_OUT := ADR(MQTT_IN_OUT));
	testPiublish[10].SetMqttInOut(MQTT_IN_OUT := ADR(MQTT_IN_OUT));
	testPiublish[11].SetMqttInOut(MQTT_IN_OUT := ADR(MQTT_IN_OUT));
	testPiublish[12].SetMqttInOut(MQTT_IN_OUT := ADR(MQTT_IN_OUT));
	testPiublish[13].SetMqttInOut(MQTT_IN_OUT := ADR(MQTT_IN_OUT));
	testPiublish[14].SetMqttInOut(MQTT_IN_OUT := ADR(MQTT_IN_OUT));
	testPiublish[15].SetMqttInOut(MQTT_IN_OUT := ADR(MQTT_IN_OUT));
	testPiublish[16].SetMqttInOut(MQTT_IN_OUT := ADR(MQTT_IN_OUT));
	testPiublish[17].SetMqttInOut(MQTT_IN_OUT := ADR(MQTT_IN_OUT));
	sub1.SetMqttInOut(MQTT_IN_OUT:= ADR(MQTT_IN_OUT));
	sub2.SetMqttInOut(MQTT_IN_OUT:= ADR(MQTT_IN_OUT));
	sub3.SetMqttInOut(MQTT_IN_OUT:= ADR(MQTT_IN_OUT));
	//Testtopic();
	FOR i := 0 TO 90 DO
		CommonTypesAndFunctions.concat(s1:= ADR(s1), s2:= ADR(sa));
		CommonTypesAndFunctions.concat(s1:= ADR(s1), s2:= ADR('/'));
		CommonTypesAndFunctions.concat(s1:= ADR(s1), s2:= ADR(sb));
		CommonTypesAndFunctions.concat(s1:= ADR(s1), s2:= ADR('/'));
	END_FOR
		FOR i := 0 TO 10 DO
		CommonTypesAndFunctions.concat(s1:= ADR(s2), s2:= ADR(sc));
		CommonTypesAndFunctions.concat(s1:= ADR(s2), s2:= ADR('/'));
		CommonTypesAndFunctions.concat(s1:= ADR(s2), s2:= ADR(sd));
		CommonTypesAndFunctions.concat(s1:= ADR(s2), s2:= ADR('/'));
	END_FOR
	FOR i := 0 TO bSize DO
		b1[i] := UDINT_TO_BYTE(i);
	END_FOR
END_IF

FOR i := 0 TO 20 DO
	CountSucsess[i] := testPiublish[i].CountSend;
END_FOR

TestLen := CommonTypesAndFunctions.len(str:= ADR(''));
TestLen := CommonTypesAndFunctions.len(str:= ADR('a'));
TestLen := CommonTypesAndFunctions.len(str:= ADR('aa'));

//	TestSubscribe();
(*
sub1(
	Subscribe:= con, 
	Topic:= ADR(s2), 
	QoSSubscribe:= 2,
	Recived => longRecived,
	ExpectingString := TRUE
	 );
sub2(
	Subscribe:= TestLongSubscribe, 
	Topic:= ADR(s1), 
	QoSSubscribe:= 2 ,
	Recived => recived1,
	ExpectingString := TRUE
	 );
sub3(
	Subscribe:= SubscribeForBigPaket, 
	Topic:= ADR('#'), 
	QoSSubscribe:= 2 ,
	Recived => recived2,
	ExpectingString := FALSE
	 );
IF recived1 THEN
	i:=i;
	ReciveData[reciveIndex].MqttPayload := sub1.PayloadString^;
	ReciveData[reciveIndex].MqttTopic := sub1.TopicOut^;
	reciveIndex := reciveIndex + 1;
	IF reciveIndex > 100 THEN
		reciveIndex := 0;
	END_IF
END_IF*)
testPiublish[17](
	Topic:= ADR(s1), 
	Payload:= ADR(b1), 
	QoSIn:= qos, 
	MRetain:= MQTTretain, 
	send := testTimeBigPayload.Q,
	PayloadLength :=  3654,
	PublishAsString := FALSE
	);
testPiublish[16](
	Topic:= ADR(s1), 
	PayloadString:= ADR(s2), 
	QoSIn:= qos, 
	MRetain:= MQTTretain, 
	send := testTimeBigPublish.Q, 
	PublishAsString := TRUE
	);
testPiublish[0](
	Topic:= ADR('test/topic veryyyyyyyyyyyyyyyyyyyyyyyyyyyyyyyyyyyyyyyyyyyyyyyyyyyyyyyyyyyyyyyyyyyyyyyyyyyyyyyyyyyyyyyyyyyyyyyyyyyyyyyyyyyyyyyyyy big topic/1'), 
	PayloadString:= ADR('test pi1'), 
	QoSIn:= qos, 
	MRetain:= MQTTretain, 
	send := testtime.Q,
	PublishAsString := TRUE 
	);
	
testPiublish[1](
	Topic:= ADR('test/topic veryyyyyyyyyyyyyyyyyyyyyyyyyyyyyyyyyyyyyyyyyyyyyyyyyyyyyyyyyyyyyyyyyyyyyyyyyyyyyyyyyyyyyyyyyyyyyyyyyyyyyyyyyyyyyyyyyy big topic/2'), 
	PayloadString:= ADR('test pi2'), 
	QoSIn:= qos, 
	MRetain:= MQTTretain, 
	send := testtime.Q,
	PublishAsString := TRUE 
	);
testPiublish[2](
	Topic:= ADR('test/topic veryyyyyyyyyyyyyyyyyyyyyyyyyyyyyyyyyyyyyyyyyyyyyyyyyyyyyyyyyyyyyyyyyyyyyyyyyyyyyyyyyyyyyyyyyyyyyyyyyyyyyyyyyyyyyyyyyy big topic/3'), 
	PayloadString:= ADR('test pi3'), 
	QoSIn:= qos, 
	MRetain:= MQTTretain, 
	send := testtime.Q,
	PublishAsString := TRUE 
	);
testPiublish[3](
	Topic:= ADR('test/topic veryyyyyyyyyyyyyyyyyyyyyyyyyyyyyyyyyyyyyyyyyyyyyyyyyyyyyyyyyyyyyyyyyyyyyyyyyyyyyyyyyyyyyyyyyyyyyyyyyyyyyyyyyyyyyyyyyy big topic/4'), 
	PayloadString:= ADR('test pi4'), 
	QoSIn:= qos, 
	MRetain:= MQTTretain, 
	send := testtime.Q, 
	PublishAsString := TRUE
	);
testPiublish[4](
	Topic:= ADR('test/topic veryyyyyyyyyyyyyyyyyyyyyyyyyyyyyyyyyyyyyyyyyyyyyyyyyyyyyyyyyyyyyyyyyyyyyyyyyyyyyyyyyyyyyyyyyyyyyyyyyyyyyyyyyyyyyyyyyy big topic/5'), 
	PayloadString:= ADR('test pi5'), 
	QoSIn:= qos, 
	MRetain:= MQTTretain, 
	send := testtime.Q, 
	PublishAsString := TRUE
	);
testPiublish[5](
	Topic:= ADR('test/topic veryyyyyyyyyyyyyyyyyyyyyyyyyyyyyyyyyyyyyyyyyyyyyyyyyyyyyyyyyyyyyyyyyyyyyyyyyyyyyyyyyyyyyyyyyyyyyyyyyyyyyyyyyyyyyyyyyy big topic/6'), 
	PayloadString:= ADR('test pi6'), 
	QoSIn:= qos, 
	MRetain:= MQTTretain, 
	send := testtime.Q, 
	PublishAsString := TRUE
	);
testPiublish[6](
	Topic:= ADR('test/topic veryyyyyyyyyyyyyyyyyyyyyyyyyyyyyyyyyyyyyyyyyyyyyyyyyyyyyyyyyyyyyyyyyyyyyyyyyyyyyyyyyyyyyyyyyyyyyyyyyyyyyyyyyyyyyyyyyy big topic/7'), 
	PayloadString:= ADR('test pi7'), 
	QoSIn:= qos, 
	MRetain:= MQTTretain, 
	send := testtime.Q, 
	PublishAsString := TRUE
	);
testPiublish[7](
	Topic:= ADR('test/topic veryyyyyyyyyyyyyyyyyyyyyyyyyyyyyyyyyyyyyyyyyyyyyyyyyyyyyyyyyyyyyyyyyyyyyyyyyyyyyyyyyyyyyyyyyyyyyyyyyyyyyyyyyyyyyyyyyy big topic/8'), 
	PayloadString:= ADR('test pi8'), 
	QoSIn:= qos, 
	MRetain:= MQTTretain, 
	send := testtime.Q, 
	PublishAsString := TRUE
	);
testPiublish[8](
	Topic:= ADR('test/topic veryyyyyyyyyyyyyyyyyyyyyyyyyyyyyyyyyyyyyyyyyyyyyyyyyyyyyyyyyyyyyyyyyyyyyyyyyyyyyyyyyyyyyyyyyyyyyyyyyyyyyyyyyyyyyyyyyy big topic/9'), 
	PayloadString:= ADR('test pi9'), 
	QoSIn:= qos, 
	MRetain:= MQTTretain, 
	send := testtime.Q, 
	PublishAsString := TRUE
	);
testPiublish[9](
	Topic:= ADR('test/topic veryyyyyyyyyyyyyyyyyyyyyyyyyyyyyyyyyyyyyyyyyyyyyyyyyyyyyyyyyyyyyyyyyyyyyyyyyyyyyyyyyyyyyyyyyyyyyyyyyyyyyyyyyyyyyyyyyy big topic/10'), 
	PayloadString:= ADR('test pi10'), 
	QoSIn:= qos, 
	MRetain:= MQTTretain, 
	send := testtime.Q, 
	PublishAsString := TRUE
	);
testPiublish[10](
	Topic:= ADR('test/topic veryyyyyyyyyyyyyyyyyyyyyyyyyyyyyyyyyyyyyyyyyyyyyyyyyyyyyyyyyyyyyyyyyyyyyyyyyyyyyyyyyyyyyyyyyyyyyyyyyyyyyyyyyyyyyyyyyy big topic/11'), 
	PayloadString:= ADR('test pi11'), 
	QoSIn:= qos, 
	MRetain:= MQTTretain, 
	send := testtime.Q, 
	PublishAsString := TRUE
	);
testPiublish[11](
	Topic:= ADR('test/topic veryyyyyyyyyyyyyyyyyyyyyyyyyyyyyyyyyyyyyyyyyyyyyyyyyyyyyyyyyyyyyyyyyyyyyyyyyyyyyyyyyyyyyyyyyyyyyyyyyyyyyyyyyyyyyyyyyy big topic/12'), 
	PayloadString:= ADR('test pi12'), 
	QoSIn:= qos, 
	MRetain:= MQTTretain, 
	send := testtime.Q, 
	PublishAsString := TRUE
	);
testPiublish[12](
	Topic:= ADR('test/topic veryyyyyyyyyyyyyyyyyyyyyyyyyyyyyyyyyyyyyyyyyyyyyyyyyyyyyyyyyyyyyyyyyyyyyyyyyyyyyyyyyyyyyyyyyyyyyyyyyyyyyyyyyyyyyyyyyy big topic/13'), 
	PayloadString:= ADR('test pi13'), 
	QoSIn:= qos, 
	MRetain:= MQTTretain, 
	send := testtime.Q, 
	PublishAsString := TRUE
	);
testPiublish[13](
	Topic:= ADR('test/topic veryyyyyyyyyyyyyyyyyyyyyyyyyyyyyyyyyyyyyyyyyyyyyyyyyyyyyyyyyyyyyyyyyyyyyyyyyyyyyyyyyyyyyyyyyyyyyyyyyyyyyyyyyyyyyyyyyy big topic/14'), 
	PayloadString:= ADR('test pi14'), 
	QoSIn:= qos, 
	MRetain:= MQTTretain, 
	send := testtime.Q, 
	PublishAsString := TRUE
	);
testPiublish[14](
	Topic:= ADR('test/topic veryyyyyyyyyyyyyyyyyyyyyyyyyyyyyyyyyyyyyyyyyyyyyyyyyyyyyyyyyyyyyyyyyyyyyyyyyyyyyyyyyyyyyyyyyyyyyyyyyyyyyyyyyyyyyyyyyy big topic/15'), 
	PayloadString:= ADR('test pi15'), 
	QoSIn:= qos, 
	MRetain:= MQTTretain, 
	send := testtime.Q, 
	PublishAsString := TRUE
	);
testPiublish[15](
	Topic:= ADR('test/topic veryyyyyyyyyyyyyyyyyyyyyyyyyyyyyyyyyyyyyyyyyyyyyyyyyyyyyyyyyyyyyyyyyyyyyyyyyyyyyyyyyyyyyyyyyyyyyyyyyyyyyyyyyyyyyyyyyy big topic/16'), 
	PayloadString:= ADR('test pi16'), 
	QoSIn:= qos, 
	MRetain:= MQTTretain, 
	send := testtime.Q, 
	PublishAsString := TRUE
	);



(*
MQTT(
	MQTT_INFO:= MQTT_INFO, 
	MQTT_IN_OUT:= MQTT_IN_OUT, 
	ENABLE:= TRUE, 
	URL:= 'test.mosquitto.org:1883', 
	TIMEOUT:= T#5S, 
	ERROR_C=> ERROR_C, 
	ERROR_T=> ERROR_T);
	*)
	(*
	MQTT(
	MQTT_INFO:= MQTT_INFO, 
	MQTT_IN_OUT:= MQTT_IN_OUT, 
	ENABLE:= enable, 
	URL:= 'localhost:1883', 
	TIMEOUT:= T#5S, 
	ERROR_C=> ERROR_C, 
	ERROR_T=> ERROR_T);
	*)



MQTT(
	MQTT_INFO:= MQTT_INFO, 
	MQTT_IN_OUT:= MQTT_IN_OUT, 
	ENABLE:= enable, 
	URL:= 'windows-10-pro:1883', 
	TIMEOUT:= T#5S, 
	ERROR_C=> ERROR_C, 
	ERROR_T=> ERROR_T);

          
END_FUNCTION_BLOCK

FUNCTION_BLOCK TestMqttTLS
  VAR
    MQTT : HANDLE_MQTT;
    MQTT_INFO : MQTT_INFO;
    MQTT_IN_OUT : MQTT_IN_OUT;
    ERROR_C : DWORD;
    ERROR_T : BYTE;
    testPiublish : ARRAY[0..100] OF MQTTPublish;  (* testPiublish: SD_MQTT.MQTTPublish; *)
    init : BOOL := FALSE;
    sendTest : BOOL;
    testtime : ton;
    i : UINT;
    qos : QoS := 2;
    sub1 : MQTTSubscribe;
    sub2 : MQTTSubscribe;
    con : BOOL;
    recived : BOOL;  (* Testtopic:SD_MQTT.TestcaseCheckTopivValid; TestSubscribe:SD_MQTT.TestSubscribe; *)
    CountSucsess : ARRAY[0..100] OF ULINT;
    MQTTretain : BOOL := TRUE;
    enable : BOOL;
    ReciveData : ARRAY[0..100] OF RECIVE_PAKET;
    reciveIndex : INT;
    testTls : BOOL := TRUE;
    TLS_CONFIG : CommonTypesAndFunctions.TLS_CONFIG;
  END_VAR

            MQTT_IN_OUT.ClientID :='testCodesys';
//MQTT_IN_OUT.PORT := 1883;
//MQTT_IN_OUT.URL := 'test.mosquitto.org';

testtime(IN:= NOT testtime.Q AND sendTest, PT:= T#100MS);
//testtime(IN:= NOT testtime.Q AND sendTest, PT:= T#10S);
IF NOT init THEN
	init := TRUE;
	testPiublish[0].SetMqttInOut(MQTT_IN_OUT := ADR(MQTT_IN_OUT));
	testPiublish[1].SetMqttInOut(MQTT_IN_OUT := ADR(MQTT_IN_OUT));
	testPiublish[2].SetMqttInOut(MQTT_IN_OUT := ADR(MQTT_IN_OUT));
	testPiublish[3].SetMqttInOut(MQTT_IN_OUT := ADR(MQTT_IN_OUT));
	testPiublish[4].SetMqttInOut(MQTT_IN_OUT := ADR(MQTT_IN_OUT));
	testPiublish[5].SetMqttInOut(MQTT_IN_OUT := ADR(MQTT_IN_OUT));
	testPiublish[6].SetMqttInOut(MQTT_IN_OUT := ADR(MQTT_IN_OUT));
	testPiublish[7].SetMqttInOut(MQTT_IN_OUT := ADR(MQTT_IN_OUT));
	testPiublish[8].SetMqttInOut(MQTT_IN_OUT := ADR(MQTT_IN_OUT));
	testPiublish[9].SetMqttInOut(MQTT_IN_OUT := ADR(MQTT_IN_OUT));
	testPiublish[10].SetMqttInOut(MQTT_IN_OUT := ADR(MQTT_IN_OUT));
	testPiublish[11].SetMqttInOut(MQTT_IN_OUT := ADR(MQTT_IN_OUT));
	testPiublish[12].SetMqttInOut(MQTT_IN_OUT := ADR(MQTT_IN_OUT));
	testPiublish[13].SetMqttInOut(MQTT_IN_OUT := ADR(MQTT_IN_OUT));
	testPiublish[14].SetMqttInOut(MQTT_IN_OUT := ADR(MQTT_IN_OUT));
	testPiublish[15].SetMqttInOut(MQTT_IN_OUT := ADR(MQTT_IN_OUT));
	sub1.SetMqttInOut(MQTT_IN_OUT:= ADR(MQTT_IN_OUT));
	sub2.SetMqttInOut(MQTT_IN_OUT:= ADR(MQTT_IN_OUT));
	//Testtopic();
	
	MQTT_IN_OUT.TLS_CONFIG := ADR(TLS_CONFIG);

END_IF

FOR i := 0 TO 20 DO
	CountSucsess[i] := testPiublish[i].CountSend;
END_FOR

//	TestSubscribe();
(*
sub1(
	Subscribe:= con, 
	Topic:= ADR('test/#'), 
	QoSSubscribe:= 2 ,
	Recived => recived,
	ExpectingString := TRUE
	 );
	 
sub2(
	Subscribe:= con, 
	Topic:= ADR('#'), 
	QoSSubscribe:= 2 ,
	Recived => recived,
	ExpectingString := TRUE
	 );
IF recived THEN
	i:=i;
	ReciveData[reciveIndex].MqttPayload := sub1.PayloadString^;
	ReciveData[reciveIndex].MqttTopic := sub1.TopicOut^;
	reciveIndex := reciveIndex + 1;
	IF reciveIndex > 100 THEN
		reciveIndex := 0;
	END_IF
END_IF*)
testPiublish[0](
	Topic:= ADR('test/topic veryyyyyyyyyyyyyyyyyyyyyyyyyyyyyyyyyyyyyyyyyyyyyyyyyyyyyyyyyyyyyyyyyyyyyyyyyyyyyyyyyyyyyyyyyyyyyyyyyyyyyyyyyyyyyyyyyy big topic/1'), 
	PayloadString:= ADR('test pi1'), 
	QoSIn:= qos, 
	MRetain:= MQTTretain, 
	send := testtime.Q,
	PublishAsString := TRUE 
	);
	
testPiublish[1](
	Topic:= ADR('test/topic veryyyyyyyyyyyyyyyyyyyyyyyyyyyyyyyyyyyyyyyyyyyyyyyyyyyyyyyyyyyyyyyyyyyyyyyyyyyyyyyyyyyyyyyyyyyyyyyyyyyyyyyyyyyyyyyyyy big topic/2'), 
	PayloadString:= ADR('test pi2'), 
	QoSIn:= qos, 
	MRetain:= MQTTretain, 
	send := testtime.Q,
	PublishAsString := TRUE 
	);
testPiublish[2](
	Topic:= ADR('test/topic veryyyyyyyyyyyyyyyyyyyyyyyyyyyyyyyyyyyyyyyyyyyyyyyyyyyyyyyyyyyyyyyyyyyyyyyyyyyyyyyyyyyyyyyyyyyyyyyyyyyyyyyyyyyyyyyyyy big topic/3'), 
	PayloadString:= ADR('test pi3'), 
	QoSIn:= qos, 
	MRetain:= MQTTretain, 
	send := testtime.Q,
	PublishAsString := TRUE 
	);
testPiublish[3](
	Topic:= ADR('test/topic veryyyyyyyyyyyyyyyyyyyyyyyyyyyyyyyyyyyyyyyyyyyyyyyyyyyyyyyyyyyyyyyyyyyyyyyyyyyyyyyyyyyyyyyyyyyyyyyyyyyyyyyyyyyyyyyyyy big topic/4'), 
	PayloadString:= ADR('test pi4'), 
	QoSIn:= qos, 
	MRetain:= MQTTretain, 
	send := testtime.Q, 
	PublishAsString := TRUE
	);
testPiublish[4](
	Topic:= ADR('test/topic veryyyyyyyyyyyyyyyyyyyyyyyyyyyyyyyyyyyyyyyyyyyyyyyyyyyyyyyyyyyyyyyyyyyyyyyyyyyyyyyyyyyyyyyyyyyyyyyyyyyyyyyyyyyyyyyyyy big topic/5'), 
	PayloadString:= ADR('test pi5'), 
	QoSIn:= qos, 
	MRetain:= MQTTretain, 
	send := testtime.Q, 
	PublishAsString := TRUE
	);
testPiublish[5](
	Topic:= ADR('test/topic veryyyyyyyyyyyyyyyyyyyyyyyyyyyyyyyyyyyyyyyyyyyyyyyyyyyyyyyyyyyyyyyyyyyyyyyyyyyyyyyyyyyyyyyyyyyyyyyyyyyyyyyyyyyyyyyyyy big topic/6'), 
	PayloadString:= ADR('test pi6'), 
	QoSIn:= qos, 
	MRetain:= MQTTretain, 
	send := testtime.Q, 
	PublishAsString := TRUE
	);
testPiublish[6](
	Topic:= ADR('test/topic veryyyyyyyyyyyyyyyyyyyyyyyyyyyyyyyyyyyyyyyyyyyyyyyyyyyyyyyyyyyyyyyyyyyyyyyyyyyyyyyyyyyyyyyyyyyyyyyyyyyyyyyyyyyyyyyyyy big topic/7'), 
	PayloadString:= ADR('test pi7'), 
	QoSIn:= qos, 
	MRetain:= MQTTretain, 
	send := testtime.Q, 
	PublishAsString := TRUE
	);
testPiublish[7](
	Topic:= ADR('test/topic veryyyyyyyyyyyyyyyyyyyyyyyyyyyyyyyyyyyyyyyyyyyyyyyyyyyyyyyyyyyyyyyyyyyyyyyyyyyyyyyyyyyyyyyyyyyyyyyyyyyyyyyyyyyyyyyyyy big topic/8'), 
	PayloadString:= ADR('test pi8'), 
	QoSIn:= qos, 
	MRetain:= MQTTretain, 
	send := testtime.Q, 
	PublishAsString := TRUE
	);
testPiublish[8](
	Topic:= ADR('test/topic veryyyyyyyyyyyyyyyyyyyyyyyyyyyyyyyyyyyyyyyyyyyyyyyyyyyyyyyyyyyyyyyyyyyyyyyyyyyyyyyyyyyyyyyyyyyyyyyyyyyyyyyyyyyyyyyyyy big topic/9'), 
	PayloadString:= ADR('test pi9'), 
	QoSIn:= qos, 
	MRetain:= MQTTretain, 
	send := testtime.Q, 
	PublishAsString := TRUE
	);
testPiublish[9](
	Topic:= ADR('test/topic veryyyyyyyyyyyyyyyyyyyyyyyyyyyyyyyyyyyyyyyyyyyyyyyyyyyyyyyyyyyyyyyyyyyyyyyyyyyyyyyyyyyyyyyyyyyyyyyyyyyyyyyyyyyyyyyyyy big topic/10'), 
	PayloadString:= ADR('test pi10'), 
	QoSIn:= qos, 
	MRetain:= MQTTretain, 
	send := testtime.Q, 
	PublishAsString := TRUE
	);
testPiublish[10](
	Topic:= ADR('test/topic veryyyyyyyyyyyyyyyyyyyyyyyyyyyyyyyyyyyyyyyyyyyyyyyyyyyyyyyyyyyyyyyyyyyyyyyyyyyyyyyyyyyyyyyyyyyyyyyyyyyyyyyyyyyyyyyyyy big topic/11'), 
	PayloadString:= ADR('test pi11'), 
	QoSIn:= qos, 
	MRetain:= MQTTretain, 
	send := testtime.Q, 
	PublishAsString := TRUE
	);
testPiublish[11](
	Topic:= ADR('test/topic veryyyyyyyyyyyyyyyyyyyyyyyyyyyyyyyyyyyyyyyyyyyyyyyyyyyyyyyyyyyyyyyyyyyyyyyyyyyyyyyyyyyyyyyyyyyyyyyyyyyyyyyyyyyyyyyyyy big topic/12'), 
	PayloadString:= ADR('test pi12'), 
	QoSIn:= qos, 
	MRetain:= MQTTretain, 
	send := testtime.Q, 
	PublishAsString := TRUE
	);
testPiublish[12](
	Topic:= ADR('test/topic veryyyyyyyyyyyyyyyyyyyyyyyyyyyyyyyyyyyyyyyyyyyyyyyyyyyyyyyyyyyyyyyyyyyyyyyyyyyyyyyyyyyyyyyyyyyyyyyyyyyyyyyyyyyyyyyyyy big topic/13'), 
	PayloadString:= ADR('test pi13'), 
	QoSIn:= qos, 
	MRetain:= MQTTretain, 
	send := testtime.Q, 
	PublishAsString := TRUE
	);
testPiublish[13](
	Topic:= ADR('test/topic veryyyyyyyyyyyyyyyyyyyyyyyyyyyyyyyyyyyyyyyyyyyyyyyyyyyyyyyyyyyyyyyyyyyyyyyyyyyyyyyyyyyyyyyyyyyyyyyyyyyyyyyyyyyyyyyyyy big topic/14'), 
	PayloadString:= ADR('test pi14'), 
	QoSIn:= qos, 
	MRetain:= MQTTretain, 
	send := testtime.Q, 
	PublishAsString := TRUE
	);
testPiublish[14](
	Topic:= ADR('test/topic veryyyyyyyyyyyyyyyyyyyyyyyyyyyyyyyyyyyyyyyyyyyyyyyyyyyyyyyyyyyyyyyyyyyyyyyyyyyyyyyyyyyyyyyyyyyyyyyyyyyyyyyyyyyyyyyyyy big topic/15'), 
	PayloadString:= ADR('test pi15'), 
	QoSIn:= qos, 
	MRetain:= MQTTretain, 
	send := testtime.Q, 
	PublishAsString := TRUE
	);
testPiublish[15](
	Topic:= ADR('test/topic veryyyyyyyyyyyyyyyyyyyyyyyyyyyyyyyyyyyyyyyyyyyyyyyyyyyyyyyyyyyyyyyyyyyyyyyyyyyyyyyyyyyyyyyyyyyyyyyyyyyyyyyyyyyyyyyyyy big topic/16'), 
	PayloadString:= ADR('test pi16'), 
	QoSIn:= qos, 
	MRetain:= MQTTretain, 
	send := testtime.Q, 
	PublishAsString := TRUE
	);




(*
MQTT(
	MQTT_INFO:= MQTT_INFO, 
	MQTT_IN_OUT:= MQTT_IN_OUT, 
	ENABLE:= TRUE, 
	URL:= 'test.mosquitto.org:1883', 
	TIMEOUT:= T#5S, 
	ERROR_C=> ERROR_C, 
	ERROR_T=> ERROR_T);
	*)
	(*
	MQTT(
	MQTT_INFO:= MQTT_INFO, 
	MQTT_IN_OUT:= MQTT_IN_OUT, 
	ENABLE:= enable, 
	URL:= 'localhost:1883', 
	TIMEOUT:= T#5S, 
	ERROR_C=> ERROR_C, 
	ERROR_T=> ERROR_T);
	*)


IF testtls THEN
	
(*
MQTT(
	MQTT_INFO:= MQTT_INFO, 
	MQTT_IN_OUT:= MQTT_IN_OUT, 
	ENABLE:= enable, 
	URL:= 'windows-10-pro:8883', //8883 encryptet, 1883 unencryptet
	TIMEOUT:= T#5S, 
	TLS := TRUE,
	ERROR_C=> ERROR_C, 
	ERROR_T=> ERROR_T);
	*)
	MQTT(
	MQTT_INFO:= MQTT_INFO, 
	MQTT_IN_OUT:= MQTT_IN_OUT, 
	ENABLE:= enable, 
	URL:= 'test.mosquitto.org:8883', //8883 encryptet, 1883 unencryptet
	TIMEOUT:= T#5S, 
	TLS := TRUE,
	ERROR_C=> ERROR_C, 
	ERROR_T=> ERROR_T);
	
	

ELSE
MQTT(
	MQTT_INFO:= MQTT_INFO, 
	MQTT_IN_OUT:= MQTT_IN_OUT, 
	ENABLE:= enable, 
	URL:= 'test.mosquitto.org:1883', //8883 encryptet, 1883 unencryptet
	TIMEOUT:= T#5S, 
	TLS := FALSE,
	ERROR_C=> ERROR_C, 
	ERROR_T=> ERROR_T);
END_IF
          
END_FUNCTION_BLOCK

